Yaskawa INFORM job: OK_R2_O38-47,64(1)(90,180)_HARDO.JBI

/JOB
//NAME OK_R2_O38-47,64(1)(90,180)_HARDO
///FOLDERNAME X4
//POS
///NPOS 800,800,800,27,0,0
///TOOL 0
///POSTYPE PULSE
///PULSE
C00000=-90909,-97924,-91406,-33882,56334,85304
C00001=-91259,-96225,-90754,-33542,56592,85046
C00002=-89195,-70570,-78323,-22025,66185,85062
C00003=-92493,-17269,-45698,-9840,97075,81335
C00004=-91017,-18219,-43079,-10012,95177,81978
C00005=-91017,-18348,-42567,-10003,94801,82008
C00006=-91017,-18513,-41854,-9992,94286,82047
C00007=-91016,-18479,-42013,-9993,94400,82038
C00008=-90999,-21146,-43962,-9991,94233,82058
C00009=-91016,-18479,-42013,-9993,94400,82038
C00010=-92024,-18257,-41848,-9852,94294,81714
C00011=-93307,-17743,-41470,-9670,94175,81298
C00012=-92024,-17970,-43013,-9870,95146,81646
C00013=-103789,-67957,-64906,12961,58029,80477
C00014=-103344,-68399,-64680,12784,57602,80605
C00015=-103344,-68177,-63508,12869,57010,80534
C00016=-103344,-68220,-63718,12855,57117,80546
C00017=-103133,-65270,-62235,12663,57675,80699
C00018=-103344,-68220,-63718,12855,57117,80546
C00019=-102110,-68679,-63945,12230,56831,81014
C00020=-100734,-69291,-64248,11527,56502,81539
C00021=-102110,-68955,-65416,12130,57578,81100
C00022=-83930,-36393,-48077,-21091,64166,86746
C00023=-83530,-35162,-44070,-21603,62556,87219
C00024=-83530,-35090,-42657,-21762,61780,87376
C00025=-83530,-35104,-42903,-21736,61913,87350
C00026=-83323,-32550,-41219,-21780,62224,87371
C00027=-83530,-35104,-42903,-21736,61913,87350
C00028=-84416,-35012,-42843,-21317,61693,87037
C00029=-85758,-34937,-42794,-20674,61360,86560
C00030=-84416,-35012,-42843,-21317,61693,87037
C00031=-98607,9794,-21494,8158,96572,85590
C00032=-98154,8993,-20894,8080,95751,85685
C00033=-98154,8801,-20162,8070,95209,85650
C00034=-98154,8841,-20318,8071,95323,85660
C00035=-98340,6335,-22513,8097,95402,85603
C00036=-98154,8841,-20318,8071,95323,85660
C00037=-97649,8538,-20585,8003,95283,85823
C00038=-96706,8027,-21034,7872,95207,86128
C00039=-97649,8860,-21759,8020,96163,85880
C00040=-91418,16997,-18664,7186,97864,88018
C00041=-81575,50041,17092,-6735,115955,80813
C00042=-84341,50404,17488,-7249,115666,79799
C00043=-84633,49569,18016,-7267,114894,79739
C00044=-84633,49489,18537,-7242,114535,79763
C00045=-84633,49518,18343,-7250,114668,79755
C00046=-84609,54795,24149,-7190,113816,79818
C00047=-84609,54766,24403,-7179,113647,79829
C00048=-84663,51666,20976,-7222,114154,79777
C00049=-84658,51948,21286,-7218,114109,79782
C00050=-84658,51915,21548,-7206,113932,79794
C00051=-84658,51950,21266,-7218,114122,79782
C00052=-84668,56412,26217,-7173,113374,79826
C00053=-84668,56378,26569,-7158,113142,79841
C00054=-84634,53730,23622,-7179,113595,79825
C00055=-84637,55494,23519,-7242,114557,79761
C00056=-81397,31619,-5447,10992,111497,83226
C00057=-81473,32242,-2198,10850,109860,83040
C00058=-81473,31956,-1216,10793,109121,82971
C00059=-81473,32044,-1532,10810,109358,82993
C00060=-81453,37801,4324,10764,108721,82941
C00061=-81453,37706,4697,10744,108448,82916
C00062=-81443,35181,2108,10765,108737,82946
C00063=-81447,36511,1500,10844,109776,83041
C00064=-95159,59700,8174,10738,119151,79045
C00065=-82349,25617,-23576,-8938,79907,82210
C00066=-85481,26023,-25062,-8026,81022,81034
C00067=-85695,25195,-23613,-7939,79706,81051
C00068=-85695,24472,-22838,-7959,78866,81106
C00069=-85695,24604,-22984,-7954,79022,81095
C00070=-85639,26782,-20858,-7986,78839,81125
C00071=-85695,24604,-22984,-7954,79022,81095
C00072=-86173,38935,-12977,-7015,88429,87162
C00073=-85344,38540,-13390,-7315,88547,87404
C00074=-86172,38929,-12971,-7015,88439,87166
C00075=-84007,53583,-39,-17366,95072,84572
C00076=-84007,52813,643,-17337,94292,84683
C00077=-84007,52406,1031,-17322,93863,84745
C00078=-84007,52527,916,-17328,93991,84727
C00079=-84079,50201,-1661,-17319,94351,84652
C00080=-84007,52527,916,-17328,93991,84727
C00081=-84889,52670,1073,-17081,93801,84474
C00082=-85681,52912,1343,-16856,93611,84250
C00083=-84889,53509,304,-17110,94667,84353
C00084=-82262,58897,13828,-12408,108012,82136
C00085=-83953,58737,25467,-6224,116924,79977
C00086=-84346,-10282,-49110,5038,88729,85099
C00087=-83106,-20728,-52489,-22212,92643,80661
C00088=-106659,-18282,-50653,-15937,87636,73637
C00089=-135463,84611,26036,-8427,98138,63561
C00090=-134711,78652,30015,-19475,126025,58919
C00091=-134415,83458,36943,-18891,124399,59387
C00092=-134415,83178,37391,-18788,124001,59464
C00093=-134415,82845,37969,-18663,123504,59559
C00094=-134415,83107,37513,-18763,123898,59484
C00095=-133823,86478,41707,-18417,123218,59859
C00096=-133823,86166,42311,-18294,122713,59953
C00097=-134051,84793,40603,-18428,122994,59806
C00098=-133823,86534,41603,-18437,123307,59843
C00099=-130836,86678,38865,-21284,122414,55409
C00100=-135463,84611,26036,-8427,98138,63561
C00101=-106659,-18282,-50653,-15937,87636,73637
C00102=-89310,-122172,-106686,-13361,50676,45199
C00103=-123165,-113898,-119110,19125,43336,-19368
C00104=-123668,-102412,-109547,19577,43467,-19587
C00105=-131184,63359,57441,15233,67840,-18691
C00106=-122068,78147,74274,12505,69533,-15106
C00107=-122051,87849,89370,12875,65325,-15559
C00108=-122051,89227,92048,12969,64408,-15664
C00109=-122316,85057,86118,12868,65923,-15592
C00110=-122667,82911,83414,12880,66527,-15655
C00111=-122667,83831,85320,12946,65844,-15732
C00112=-122426,86931,89254,12983,65000,-15737
C00113=-122963,79390,78884,12845,67528,-15654
C00114=-130632,64185,60223,15235,66493,-18662
C00115=-131662,58983,54996,15425,67212,-18954
C00116=-131668,55339,42428,14901,72880,-18222
C00117=-146861,-92393,-105699,36485,53490,-27620
C00118=-148000,-101656,-114811,36865,54640,-27702
C00119=-148000,-101656,-114811,36865,54640,-27702
C00120=-148000,-101656,-114811,36865,54640,-27702
C00121=-159496,-161049,-136264,30615,73499,-21221
C00122=-103228,-122632,-133352,-7038,92284,-523
C00123=-103228,-122632,-133352,-7038,92284,-523
C00124=-103228,-124480,-131601,-7026,90271,-411
C00125=-103391,-121920,-131082,-6996,91247,-517
C00126=-103853,-115329,-128981,-6922,93290,-780
C00127=-103391,-120798,-132087,-7006,92433,-583
C00128=-104641,-114737,-130152,-6774,94243,-1084
C00129=-104641,-114737,-130152,-6774,94243,-1084
C00130=-104641,-116137,-129119,-6762,92896,-1012
C00131=-104641,-115940,-129279,-6764,93095,-1023
C00132=-105111,-108950,-126961,-6694,95208,-1287
C00133=-104576,-115792,-130426,-6785,93876,-1044
C00134=-103741,-127928,-135528,-6927,90867,-609
C00135=-103741,-127928,-135528,-6927,90867,-609
C00136=-103741,-127928,-135528,-6927,90867,-609
C00137=-103865,-116944,-129962,-6921,93061,-771
C00138=-103865,-118485,-128547,-6909,91408,-679
C00139=-103865,-118011,-129031,-6913,91946,-709
C00140=-104350,-111197,-126797,-6823,94018,-978
C00141=-103645,-119716,-131347,-6963,92509,-670
C00142=-126331,-111187,-127566,-2170,93341,-7936
C00143=-126314,-110675,-127191,-2173,93374,-7931
C00144=-126314,-111741,-126360,-2171,92316,-7913
C00145=-126314,-111248,-126762,-2172,92816,-7922
C00146=-126152,-104604,-124481,-2216,94828,-7909
C00147=-126314,-111061,-126906,-2173,93001,-7925
C00148=-125902,-111149,-126935,-2263,92984,-7794
C00149=-132196,-109284,-126305,2386,93568,-14490
C00150=-132014,-110397,-125220,2342,92324,-14457
C00151=-132014,-111538,-124094,2340,91046,-14481
C00152=-132014,-110972,-124684,2340,91699,-14468
C00153=-131346,-109003,-124013,2196,92280,-14246
C00154=-132122,-112463,-125993,2364,91740,-14502
C00155=-130696,-128652,-136015,2037,89553,-14081
C00156=-130696,-128652,-136015,2037,89553,-14081
C00157=-134573,-129962,-127961,2886,84044,-15460
C00158=-135247,-123905,-124729,3029,85191,-15657
C00159=-135247,-124242,-122895,3032,83891,-15687
C00160=-135059,-121526,-122583,2986,85086,-15595
C00161=-134621,-115318,-120572,2888,87018,-15405
C00162=-135273,-124345,-124575,3033,84868,-15671
C00163=-101634,-140552,-130463,-4330,80438,-4385
C00164=-100831,-135445,-127742,-4507,81431,-4148
C00165=-100831,-135220,-126147,-4516,80567,-4118
C00166=-100831,-135304,-126661,-4513,80840,-4129
C00167=-101541,-127818,-124438,-4340,83274,-4455
C00168=-100689,-136992,-128168,-4541,80909,-4084
C00169=-101700,-117063,-135109,-4321,95328,-4920
C00170=-101700,-117063,-135109,-4321,95328,-4920
C00171=-107464,-106510,-121453,-3057,92107,-6652
C00172=-105693,-105772,-119256,-3437,91202,-6062
C00173=-105693,-106748,-117862,-3435,89847,-6024
C00174=-105693,-106325,-118509,-3436,90460,-6041
C00175=-104724,-99451,-116018,-3652,92493,-5788
C00176=-105563,-106984,-120499,-3466,91350,-6023
C00177=-97637,-124436,-133710,-5150,90918,-3458
C00178=-101700,-117063,-135109,-4321,95328,-4920
C00179=-101700,-117063,-135109,-4321,95328,-4920
C00180=-113885,-115939,-123860,-1658,88568,-8649
C00181=-113885,-115976,-123799,-1658,88510,-8649
C00182=-113885,-116503,-122835,-1658,87648,-8639
C00183=-113928,-115223,-122529,-1647,88114,-8658
C00184=-114061,-111130,-121156,-1620,89368,-8717
C00185=-113613,-117192,-124203,-1715,88138,-8556
C00186=-77135,-109099,-124316,-9289,94737,2930
C00187=-77964,-100968,-118468,-9143,95217,2626
C00188=-77964,-101677,-117713,-9127,94398,2685
C00189=-77964,-101560,-117850,-9129,94540,2675
C00190=-78928,-97543,-116360,-8967,95572,2290
C00191=-77908,-100245,-119438,-9173,96179,2574
C00192=-71973,-123086,-130703,-10190,92110,4818
C00193=-61369,-106979,-129386,18745,110548,-43775
C00194=-54050,-118433,-122678,29834,105379,-66043
C00195=-54050,-118432,-122677,29849,105379,-66042
C00196=-52380,-128849,-120518,29019,98947,-67079
C00197=-52380,-128559,-118965,28945,98241,-67262
C00198=-52380,-128751,-119946,28990,98681,-67146
C00199=-50245,-132811,-121152,28917,96763,-66805
C00200=-52380,-128751,-119946,28990,98681,-67146
C00201=-49374,-119498,-117890,29381,100712,-65454
C00202=-49135,-119946,-117683,29342,100317,-65463
C00203=-49135,-119959,-116418,29258,99629,-65643
C00204=-49135,-119963,-116925,29289,99902,-65571
C00205=-47420,-122909,-117861,29192,98489,-65269
C00206=-49767,-118756,-118042,29437,101266,-65461
C00207=-58824,-127197,-127906,29549,105900,-67783
C00208=-58824,-127197,-127906,29549,105900,-67783
C00209=-55789,-138532,-125635,28743,98511,-68512
C00210=-54845,-137144,-123724,28738,97781,-68329
C00211=-54845,-136558,-122036,28679,97131,-68490
C00212=-54845,-136878,-122937,28709,97474,-68406
C00213=-52687,-141381,-124200,28678,95380,-68093
C00214=-56052,-135036,-125386,28893,100051,-68223
C00215=-56052,-135036,-125386,28893,100051,-68223
C00216=-54923,-136926,-123517,28734,97796,-68355
C00217=-54923,-136449,-122129,28684,97260,-68488
C00218=-54923,-136715,-122887,28711,97551,-68416
C00219=-52628,-141500,-124230,28677,95326,-68085
C00220=-54923,-138669,-131970,29176,101590,-67387
C00221=-49576,-128334,-132403,27234,106270,-69223
C00222=-44922,-139442,-128392,26353,97465,-69516
C00223=-43106,-142181,-127565,26251,95168,-69348
C00224=-43106,-141292,-125343,26201,94348,-69532
C00225=-43106,-141708,-126356,26223,94717,-69449
C00226=-42222,-150085,-128620,26118,91814,-69764
C00227=-43106,-141708,-126356,26223,94717,-69449
C00228=-58006,-149727,-131155,24086,101568,-78058
C00229=-67130,-160484,-130477,19696,102779,-86761
C00230=-65656,-163702,-131169,20680,100336,-85246
C00231=-25743,-109032,-115433,27145,106620,-70118
C00232=-31386,-185321,-134069,30256,67850,-60806
C00233=-40913,-181249,-136978,30366,76641,-63974
C00234=-31337,-124593,-132531,25311,107075,-53461
C00235=-107165,-96970,-126665,-3187,100215,-6761
C00236=-107165,-106401,-121090,-3121,91950,-6553
C00237=-99006,-123912,-120398,-10471,76789,317
C00238=-104449,-120133,-119195,-8811,77334,-1598
C00239=-136314,-76901,-102772,1273,87959,-12257
C00240=-129245,-75238,-102051,-6216,89043,-4909
C00241=-138081,-104464,-122106,1833,85725,-12838
C00242=-119260,-105046,-123410,-8534,87528,-2432
C00243=-124620,-151805,-134891,-7305,72242,-3267
C00244=-124614,-151414,-134787,-7302,72378,-3273
C00245=-124612,-151215,-134734,-7300,72449,-3276
C00246=-124620,-151805,-134891,-7305,72242,-3267
C00247=-127969,-108981,-129625,-6073,90620,-5362
C00248=-128058,-112032,-130642,-6044,89675,-5344
C00249=-99990,-117497,-120264,-13536,83880,4252
C00250=-95946,-115412,-117807,-14495,84133,5598
C00251=-139069,-101671,-113062,-2900,83618,-8638
C00252=-134512,-124069,-125019,-4259,79673,-7022
C00253=-124704,-125859,-130096,-7035,82535,-3892
C00254=-99313,-127153,-133045,12119,95446,-32872
C00255=-57886,-133831,-130402,29291,103936,-67934
C00256=-55789,-138532,-125635,28743,98511,-68512
C00257=-48693,-117877,-116324,29063,104784,-69163
C00258=-50073,-120833,-117390,28223,106210,-71565
C00259=-68626,-163926,-129258,19114,104295,-87122
C00260=-70376,-133538,-127464,20847,118406,-85282
C00261=-70376,-133538,-127464,20847,118406,-85282
C00262=-57461,-97931,-109353,30188,105270,-63675
C00263=-56121,-79134,-101591,31100,116741,-68778
C00264=-90239,-137211,-122130,21625,111934,-84005
C00265=-78206,-119593,-116830,16675,122083,-90308
C00266=-77714,-101700,-117389,19308,131076,-88387
C00267=-81561,-124200,-134149,21063,125175,-90603
C00268=-103376,-109759,-132308,-3968,97270,-5504
C00269=-101634,-140552,-130463,-4330,80438,-4385
C00270=-110031,-125673,-123303,3182,83425,-15942
C00271=-90641,-116743,-120449,-11075,89773,6751
C00272=-125358,-116095,-120243,-4332,86705,-4548
C00273=-114606,-95150,-113030,-13927,98680,11559
C00274=-109678,-119625,-133746,-14623,99658,13079
C00275=-112326,-124641,-135293,-14185,97639,12436
C00276=-113675,-111285,-124420,-14007,97585,11993
C00277=-113699,-111426,-124467,-14002,97539,11990
C00278=-124004,-129907,-130136,-8507,87303,2218
C00279=-139409,-131326,-130615,456,84743,-11777
C00280=-149006,-99791,-120232,2566,94725,-14751
C00281=-149042,-99754,-120218,2574,94737,-14762
C00282=-144445,-99331,-120062,1565,94748,-13320
C00283=-148134,-92536,-117492,2386,96740,-14437
C00284=-154718,-145008,-134516,3815,80522,-16974
C00285=-155631,-143491,-134098,4008,81086,-17267
C00286=-124045,-119827,-121338,-6126,86009,-1689
C00287=-127884,-116949,-120404,-5328,86643,-2988
C00288=-148100,-95243,-112662,-980,92257,-9671
C00289=-137287,-91556,-109748,-13625,92659,296
C00290=-127829,-127486,-128792,-15513,87749,4031
C00291=-127829,-122446,-134816,-15592,93826,3264
C00292=-125285,-108995,-105645,24533,66859,-22374
C00293=-121876,-100663,-100590,22961,66967,-21017
C00294=-120611,-97454,-98556,22372,66992,-20522
C00295=-120728,-95778,-96365,22498,66572,-20652
C00296=-120611,-97454,-98556,22372,66992,-20522
C00297=-120972,-98646,-98782,22597,66650,-20731
C00298=-119814,-94892,-97816,21908,67582,-20099
C00299=-120972,-98646,-98782,22597,66650,-20731
C00300=-122255,-101873,-100811,23195,66623,-21236
C00301=-125713,-110249,-105850,24792,66512,-22621
C00302=-125414,-109454,-110952,25434,70557,-21724
C00303=-121886,-100912,-105844,23885,70668,-20357
C00304=-120575,-97642,-103795,23303,70688,-19860
C00305=-120636,-96154,-101667,23400,70203,-19982
C00306=-120575,-97642,-103795,23303,70688,-19860
C00307=-121028,-97980,-103315,23548,70382,-20093
C00308=-119871,-93906,-102218,22897,71374,-19458
C00309=-121028,-97980,-103315,23548,70382,-20093
C00310=-122351,-101230,-105354,24132,70373,-20595
C00311=-125908,-109706,-110431,25687,70298,-21973
C00312=-125468,-108852,-114009,26132,73198,-21211
C00313=-121864,-100250,-108878,24604,73277,-19846
C00314=-120523,-96969,-106822,24029,73283,-19350
C00315=-120543,-95651,-104748,24106,72739,-19471
C00316=-120523,-96969,-106822,24029,73283,-19350
C00317=-121096,-97384,-106424,24308,73024,-19616
C00318=-119937,-93066,-105230,23683,74062,-18974
C00319=-121096,-97384,-106424,24308,73024,-19616
C00320=-122450,-100644,-108468,24886,73032,-20117
C00321=-126090,-109173,-113564,26418,72994,-21493
C00322=-126107,-105383,-120588,25792,78658,-20214
C00323=-115870,-101424,-121533,-41206,90180,-3452
C00324=-115851,-106682,-115012,-41260,85065,-1433
C00325=-119242,-98694,-109765,-40357,84214,-2540
C00326=-120508,-95652,-107669,-40003,83867,-2939
C00327=-120512,-93942,-105232,-40036,83383,-2757
C00328=-120508,-95652,-107669,-40003,83867,-2939
C00329=-119976,-95300,-106376,-40178,83625,-2624
C00330=-123146,-93912,-105979,-39274,82602,-3565
C00331=-119976,-95300,-106376,-40178,83625,-2624
C00332=-118706,-98291,-108457,-40527,83992,-2228
C00333=-115305,-106116,-113657,-41413,84900,-1133
C00334=-117529,-113204,-110114,-15038,59483,16836
C00335=-119860,-102582,-104476,-13511,61010,15725
C00336=-120710,-98611,-102232,-12973,61516,15338
C00337=-120712,-96036,-99318,-13028,61058,15391
C00338=-120710,-98611,-102232,-12973,61516,15338
C00339=-120133,-97446,-101425,-13271,61707,15536
C00340=-121539,-92419,-99938,-12330,63118,14842
C00341=-120133,-97446,-101425,-13271,61707,15536
C00342=-119274,-101350,-103659,-13810,61233,15923
C00343=-116924,-111770,-109266,-15331,59803,17031
C00344=-118012,-90030,-113480,-10859,76824,11039
C00345=-121151,-43618,-104634,1145,105190,-4571
C00346=-120753,-40362,-99446,1000,103667,-4481
C00347=-120604,-39041,-97355,946,103057,-4446
C00348=-120606,-40163,-95662,941,101440,-4458
C00349=-120604,-39041,-97355,946,103057,-4446
C00350=-120772,-35445,-95769,1008,103931,-4483
C00351=-120462,-29091,-92658,908,105279,-4391
C00352=-120772,-35445,-95769,1008,103931,-4483
C00353=-120921,-36668,-97839,1062,104577,-4517
C00354=-121319,-39651,-102962,1210,106200,-4605
C00355=-108629,-121399,-122702,-16889,67135,14241
C00356=-115336,-113367,-105488,-19088,53546,18271
C00357=-117865,-102996,-100223,-17109,54980,16930
C00358=-118786,-99066,-98108,-16412,55481,16461
C00359=-118815,-96798,-95161,-16518,54853,16552
C00360=-118786,-99066,-98108,-16412,55481,16461
C00361=-119112,-97264,-98148,-16039,56331,16193
C00362=-118757,-93015,-97035,-15990,57843,16106
C00363=-119112,-97264,-98148,-16039,56331,16193
C00364=-123316,-98367,-98161,-13561,55035,14648
C00365=-126858,-97217,-97820,-11275,54872,13210
C00366=-123316,-98367,-98161,-13561,55035,14648
C00367=-122519,-102389,-100318,-14180,54451,15058
C00368=-120328,-113051,-105701,-15959,52759,16243
C00369=-124093,-110707,-95637,16539,52225,-18162
C00370=-121727,-101468,-90458,14864,53273,-16967
C00371=-120864,-97923,-88367,14268,53637,-16545
C00372=-120864,-95769,-85768,14357,53158,-16613
C00373=-120864,-97923,-88367,14268,53637,-16545
C00374=-120753,-94948,-87925,13988,54838,-16331
C00375=-119636,-91806,-87160,13170,55764,-15745
C00376=-120753,-94948,-87925,13988,54838,-16331
C00377=-121593,-98445,-90034,14553,54501,-16732
C00378=-123889,-107558,-95262,16133,53518,-17861
C00379=-123907,-109460,-104253,15319,57915,-17198
C00380=-120718,-89127,-94408,-93,103364,81793
C00381=-120702,-88967,-86044,-90,98299,81802
C00382=-120714,-92346,-83648,-90,95088,81800
C00383=-120719,-93530,-82604,-90,93837,81800
C00384=-120721,-91291,-79709,-90,93204,81799
C00385=-120719,-93530,-82604,-90,93837,81800
C00386=-120503,-94372,-82680,-81,93451,81873
C00387=-120503,-97134,-83277,-81,92401,81874
C00388=-120503,-94372,-82680,-81,93451,81873
C00389=-120501,-93212,-83739,-81,94699,81873
C00390=-120496,-89894,-86173,-82,97902,81873
C00391=-120512,-90208,-94601,-84,102927,81864
C00392=-120739,-87258,-85833,-92,99047,81789
C00393=-120752,-90752,-83510,-91,95822,81787
C00394=-120758,-91982,-82493,-91,94564,81786
C00395=-120759,-89478,-79257,-91,93861,81786
C00396=-120758,-91982,-82493,-91,94564,81786
C00397=-120462,-95334,-83503,-80,93464,81887
C00398=-120461,-97919,-84058,-79,92477,81888
C00399=-120462,-95334,-83503,-80,93464,81887
C00400=-120460,-94163,-84562,-80,94717,81887
C00401=-120456,-90813,-86994,-80,97935,81887
C00402=-121033,-93279,-128320,140,99068,-4698
C00403=-120997,-110061,-117241,128,83627,-4703
C00404=-120579,-101211,-110995,15,84330,-4566
C00405=-120424,-97983,-108548,-25,84483,-4515
C00406=-120430,-96385,-106046,-24,83763,-4517
C00407=-120424,-97983,-108548,-25,84483,-4515
C00408=-120936,-92390,-106244,111,85940,-4681
C00409=-120538,-86818,-104536,4,87751,-4552
C00410=-120936,-92390,-106244,111,85940,-4681
C00411=-121096,-95373,-108656,154,85891,-4732
C00412=-121527,-103462,-114785,270,85508,-4872
C00413=-75677,-91018,-121004,-38809,104477,-3256
C00414=-86494,-89564,-122641,-29897,102391,-4704
C00415=-121241,-108971,-117698,1136,79653,-4828
C00416=-120728,-99263,-111358,963,80734,-4651
C00417=-120539,-95742,-108880,900,81016,-4587
C00418=-120543,-94296,-106552,902,80326,-4593
C00419=-120539,-95742,-108880,900,81016,-4587
C00420=-120728,-93992,-107595,961,81127,-4647
C00421=-120728,-90301,-106424,959,82303,-4638
C00422=-120728,-93992,-107595,961,81127,-4647
C00423=-121024,-97533,-112143,1058,82109,-4735
C00424=-121551,-107098,-118478,1235,81100,-4915
C00425=-121569,-100080,-124444,1231,88376,-4850
C00426=-117898,-83225,-110918,-12916,113641,67504
C00427=-119870,-90654,-110250,-12481,109228,67312
C00428=-120686,-93336,-109842,-12338,107519,67211
C00429=-120688,-92183,-107571,-12276,106730,67294
C00430=-120686,-93336,-109842,-12338,107519,67211
C00431=-120163,-91649,-109473,-12395,108219,67318
C00432=-121681,-97188,-111137,-12239,106219,67001
C00433=-120163,-91649,-109473,-12395,108219,67318
C00434=-119359,-88923,-109851,-12543,109932,67413
C00435=-117416,-81399,-110449,-12994,114344,67589
C00436=-120617,-94125,-108136,8857,121741,88541
C00437=-120616,-94449,-107526,8800,121205,88496
C00438=-136098,-107181,-107429,16269,112846,84409
C00439=-120444,-95183,-107742,8816,120947,88541
C00440=-119761,-91680,-105499,9024,121288,-74873
C00441=-120616,-95784,-105179,-19399,105655,65758
C00442=-120617,-94769,-108163,-19676,107886,65380
C00443=-121686,-93853,-106574,-24019,104588,57765
C00444=-120617,-92780,-110041,-24421,107344,57569
C00445=-120617,-90665,-112384,-24828,109654,57058
C00446=-120619,-82046,-117525,-26421,116533,55408
C00447=-120645,-81988,-112872,-3577,88664,15070
C00448=-120614,-96077,-90479,12976,48732,-14983
C00449=-120612,-93911,-81283,13967,44304,-15634
C00450=-120612,-93390,-79613,14157,43566,-15753
C00451=-121252,-93346,-79166,14714,43437,-16096
C00452=-121500,-95247,-79374,15137,42660,-16355
C00453=-120782,-94947,-80724,14317,43483,-15851
C00454=-120611,-93982,-79716,14233,43318,-15795
C00455=-120612,-95725,-83890,13821,44941,-15536
C00456=-121326,-94847,-83951,14224,45559,-15784
C00457=-120613,-94980,-84633,13612,45776,-15407
C00458=-120613,-95388,-86250,13438,46540,-15293
C00459=-120616,-96933,-104006,-5046,49827,-739
C00460=-120616,-97132,-103061,-5097,49146,-704
C00461=-120617,-95323,-101728,-5088,49256,-711
C00462=-120871,-100699,-104338,-4972,48087,-759
C00463=-120795,-98262,-101888,-5054,47837,-712
C00464=-120618,-95198,-103493,-5003,50401,-770
C00465=-121122,-95129,-103646,-4600,50501,-986
C00466=-120617,-97030,-104927,-5009,50342,-766
C00467=-120617,-96757,-105844,-4959,51045,-801
C00468=-120618,-92718,-112658,-4589,57292,-1090
C00469=-108098,-105677,-132023,-7461,89264,328
C00470=-80455,-75739,-120669,-16714,100968,7375
C00471=-97258,-84752,-105297,-10869,90674,3530
C00472=-97358,-86422,-102930,-10833,88387,3696
C00473=-97424,-86715,-102018,-10818,87679,3736
C00474=-97216,-90521,-102980,-10875,86365,3919
C00475=-97404,-84940,-102216,-10822,88698,3655
C00476=-120617,-94266,-106774,-4665,84598,-3614
C00477=-111454,-84543,-103018,-13521,90962,7073
C00478=-109783,-86139,-104921,-12729,90791,5985
C00479=-106092,-100123,-116923,-13597,91547,7106
C00480=-102052,-116072,-128299,-14497,91044,8487
C00481=-91007,-121504,-125767,-15485,91359,21712
C00482=-120613,-95050,-86060,-3557,95049,80550
C00483=-120612,-93945,-81838,-3544,93023,80607
C00484=-121155,-91942,-79314,-3616,92478,80448
C00485=-120652,-94806,-81837,-3543,92579,80606
C00486=-120610,-90975,-79567,-3544,93151,80605
C00487=-150255,-82598,-75582,-4413,93505,70504
C00488=-122384,-91795,-77981,-11848,92227,69969
C00489=-120612,-93489,-79991,-12120,92904,70125
C00490=-120613,-94640,-84016,-12161,94749,69944
C00491=-120614,-96377,-93023,-12320,99298,69491
C00492=-120644,-125570,-121052,6784,67869,5403
C00493=-120615,-96622,-98748,12572,58745,-14095
C00494=-120615,-96643,-96984,12717,57674,-14222
C00495=-127606,-89142,-93330,20657,62312,-19456
C00496=-120926,-99715,-97034,13118,56212,-14526
C00497=-120613,-97817,-97899,12721,57634,-14225
C00498=-120615,-96818,-95655,-6616,54391,-866
C00499=-120615,-97044,-96976,-6561,55085,-910
C00500=-112093,-90513,-93108,-22044,58833,17349
C00501=-120615,-96644,-96112,-9528,53512,9485
C00502=-120615,-96653,-97679,-9416,54459,9397
C00503=-120616,-95373,-105489,-8868,59856,8934
C00504=-117333,-91440,-108817,-14098,83709,30265
C00505=-112347,-94381,-87846,-22750,99580,64599
C00506=-112329,-92021,-78548,-22454,95406,65402
C00507=-115628,-91274,-75119,-22621,92902,64661
C00508=-117255,-90241,-73175,-22718,91835,64269
C00509=-117028,-88603,-73220,-22719,92705,64185
C00510=-116923,-92272,-75451,-22697,92259,64308
C00511=-120553,-90828,-77383,15099,94128,70510
C00512=-120613,-90885,-77384,15804,94030,70628
C00513=-123770,-105111,-82751,16580,84167,79857
C00514=-124886,-104010,-85216,16560,86394,79763
C00515=-120613,-94284,-84162,15892,96365,70931
C00516=-120614,-95920,-93129,16139,100869,71526
C00517=-120649,-92160,-111225,3199,84919,49711
C00518=-120616,-97604,-99172,-11891,40402,23254
C00519=-120614,-96911,-90603,-13253,35598,24030
C00520=-120614,-96763,-89737,-13401,35153,24111
C00521=-121291,-96342,-89250,-12683,34963,23744
C00522=-119113,-97762,-90324,-15090,35268,24978
C00523=-120705,-99580,-90146,-13704,33974,24279
C00524=-121588,-95238,-86691,-12692,33949,23762
C00525=-127502,-77730,-88040,1756,56127,19882
C00526=-125086,-93679,-98074,150,54079,20822
C00527=-120613,-95818,-85653,-14108,33181,24494
C00528=-120615,-97479,-97669,-6545,55280,-923
C00529=-121580,-96410,-96097,-5967,54791,-1285
C00530=-120928,-100587,-97757,-6468,53722,-953
C00531=-120613,-98670,-98620,-6548,55254,-920
C00532=-120615,-96854,-96360,-6584,54805,-893
C00533=-120615,-97074,-97513,-6537,55399,-931
C00534=-114077,-92170,-94328,-19163,57465,15491
C00535=-120615,-97626,-97578,-9481,53904,9448
C00536=-120636,-112691,-117418,-8831,59265,10492
C00537=-120617,-94408,-109491,-7961,65698,13071
C00538=-120616,-97035,-102174,-8375,59902,13490
C00539=-120616,-97254,-100452,-8474,58742,13580
C00540=-120616,-96110,-99125,-8495,58514,13598
C00541=-120614,-98453,-101360,-8481,58685,13585
C00542=-119727,-100186,-100479,-9138,57364,14041
C00543=-120617,-96158,-99373,-8483,58642,13587
C00544=-120616,-97215,-100721,-8458,58926,13566
C00545=-120616,-96978,-102436,-8360,60091,13476
C00546=-120617,-94247,-109716,-7948,65917,13056
C00547=-120616,-96445,-103082,5252,59171,-13430
C00548=-120615,-96888,-94956,5569,53965,-13694
C00549=-120614,-96711,-93127,5642,52935,-13750
C00550=-120614,-96618,-92386,5672,52529,-13773
C00551=-119756,-94067,-91753,5051,53390,-13370
C00552=-120525,-97964,-94062,5589,52861,-13717
C00553=-120614,-96681,-92800,5656,52750,-13760
C00554=-120614,-96709,-92988,5648,52851,-13755
C00555=-120614,-96767,-93400,5632,53074,-13742
C00556=-120614,-96843,-94134,5603,53484,-13720
C00557=-120615,-96977,-95945,5531,54526,-13664
C00558=-120616,-97003,-101109,6851,58481,-13557
C00559=-120615,-97139,-99377,6934,57353,-13629
C00560=-120615,-97164,-98672,6968,56909,-13657
C00561=-119756,-94335,-97933,6375,57832,-13263
C00562=-120570,-98373,-100300,6912,57283,-13615
C00563=-120615,-97165,-99156,6946,57204,-13638
C00564=-120616,-97129,-99856,6912,57651,-13610
C00565=-120616,-96964,-101578,6829,58787,-13537
C00566=-120617,-96349,-105255,7716,61917,-13386
C00567=-120616,-96771,-103611,7804,60699,-13471
C00568=-120616,-96905,-102940,7840,60222,-13505
C00569=-119756,-93851,-102113,7266,61195,-13116
C00570=-120602,-97980,-104523,7800,60639,-13470
C00571=-120616,-96844,-103353,7819,60505,-13485
C00572=-120616,-96699,-104019,7783,60985,-13451
C00573=-120617,-96245,-105652,7696,62212,-13366
C00574=-120618,-92150,-112439,7334,68442,-12961
C00575=-130920,-122289,-127601,-23263,76296,33617
C00576=-126647,-121486,-124764,-14921,71090,19914
C00577=-118673,-117816,-113052,-9081,54805,1270
C00578=-119719,-97166,-102733,-8035,58912,525
C00579=-118944,-92090,-109805,-27006,83902,36269
C00580=-120616,-93914,-111601,-26462,83549,35758
C00581=-120617,-94475,-108119,-24525,75199,30020
C00582=-120618,-90011,-113520,-23738,94905,43572
C00583=-120617,-93534,-109718,-22404,79768,31867
C00584=-120617,-93028,-110386,-24696,84592,28860
C00585=-120617,-93859,-109223,-24523,82429,27907
C00586=-120617,-95217,-106728,-22357,73913,21133
C00587=-120616,-96198,-104144,-16550,64688,11231
C00588=-120616,-97587,-102867,-7505,58697,196
C00589=-120615,-98378,-102979,677,57412,-8649
C00590=-120615,-98092,-104435,2505,58558,-10610
C00591=-120615,-97859,-104607,2041,58746,-10113
C00592=-120615,-97689,-104685,1580,58853,-9618
C00593=-120615,-97267,-104663,-2078,59079,-5700
C00594=-122185,-96113,-104438,-1107,59504,-6297
C00595=-124417,-94235,-103728,259,60020,-7133
C00596=-120617,-96195,-105273,-2057,60007,-5718
C00597=-120617,-95777,-106468,-2039,60956,-5736
C00598=-120690,-30346,-78642,22937,64170,-21118
C00599=-120690,-30346,-78642,22937,64170,-21118
C00600=-98469,-5770,-79404,6171,73775,-13621
C00601=-73961,-64832,-115099,-11040,66386,-6438
C00602=-152983,-151482,-105999,63266,53723,19798
C00603=-133395,-32083,-56059,41211,61963,37621
C00604=-138234,23065,45169,67508,45202,44915
C00605=-136781,30072,55747,70235,43147,43411
C00606=-136213,33214,60449,71542,42329,42699
C00607=-136213,31591,57334,70422,42710,43384
C00608=-136788,30891,57778,71075,42855,42892
C00609=-134893,29619,56778,71118,41623,43172
C00610=-133284,25640,52793,70642,40733,43707
C00611=-131869,22445,49655,70246,39929,44150
C00612=-132436,19576,45433,69035,40713,44782
C00613=-133889,13007,35719,66469,42691,46136
C00614=-120930,8852,32410,71146,24358,44597
C00615=-120056,16713,42856,76185,23038,42237
C00616=-120570,20810,47735,78353,23157,41125
C00617=-120179,17981,45384,78314,22894,41190
C00618=-119718,18730,44666,76295,22791,42223
C00619=-125399,29317,56132,80433,26238,39500
C00620=-125034,24898,50699,78244,26224,40637
C00621=-126001,16678,39521,73266,27604,43020
C00622=-110893,28996,24386,6920,61269,70362
C00623=-121937,-147756,-98721,13314,47766,64479
C00624=-71720,-152863,-104081,-12596,70757,83485
C00625=-71720,-152863,-104081,-12596,70757,83485
C00626=-91982,-28216,-51992,2303,92813,79298
C00627=-105745,54824,-16277,12342,106777,76346
C00628=-79811,47197,33770,-5226,114025,80115
C00629=-80023,42119,31306,-5246,112923,80086
C00630=-80397,41231,31844,-5317,112121,79984
C00631=-80109,39795,28796,-5290,113266,80037
C00632=-80112,42618,33014,-5241,112126,80089
C00633=-81014,41143,31800,-5517,112061,79755
C00634=-81200,40698,29696,-5625,113108,79635
C00635=-82013,41869,30925,-5879,112897,79339
C00636=-81757,29065,16922,-5439,108904,79311
C00637=-82874,29136,16993,-5696,108820,78911
C00638=-83189,43833,33118,-6256,112463,78920
C00639=-80599,47195,33767,-5484,113974,79819
C00640=-80608,45992,24153,-5781,119246,79546
C00641=-80156,46426,18785,-6968,101557,41119
C00642=-78753,47274,23775,-10662,32517,-78562
C00643=-79428,-41610,-51646,-9616,33163,-79071
C00644=-79413,-40970,-42943,-11157,28217,-78271
C00645=-79779,-35257,-36372,-11029,27079,-78324
C00646=-81991,-26459,-36295,-2567,38667,-80402
C00647=-79917,-33213,-35108,-10725,27328,-78472
C00648=-79914,-35155,-35130,-11097,26361,-78286
C00649=-83153,-26286,-36175,-1364,38653,-81015
C00650=-81501,-33436,-35517,-8333,27283,-79626
C00651=-82704,-33725,-35707,-6541,27141,-80488
C00652=-84536,-24696,-36395,719,41193,-81637
C00653=-85703,-24509,-36263,1843,41226,-82218
C00654=-83984,-33203,-37030,-4447,28135,-81499
C00655=-80764,-40975,-42948,-9214,28047,-79206
C00656=-80778,-41615,-51650,-7929,33019,-79872
C00657=-86790,-31694,-78031,7959,81796,-79340
C00658=-86790,-31694,-78031,7959,81796,54010
C00659=-85481,26023,-25062,-8026,81022,81034
C00660=-85601,25422,-23671,-8007,79839,81046
C00661=-84918,26463,-20904,-8350,78751,81327
C00662=-84396,34572,-13203,-16967,82171,79029
C00663=-84396,34572,-13203,-16967,82171,79029
C00664=-86241,53458,1953,-14539,94111,75660
C00665=-83535,64450,13715,-20994,99928,87619
C00666=-86164,73511,21600,-12190,104413,87957
C00667=-86834,68614,15196,-6594,103697,88880
C00668=-86834,68614,15196,-6594,103697,88880
C00669=-86265,58182,4340,-6215,98305,89490
C00670=-84918,26463,-20904,-8350,78751,81327
C00671=-84270,25392,-25849,-8593,81276,81352
C00672=-83330,-46575,-52890,-13958,55049,-41505
C00673=-86193,-52033,-54165,-20785,79907,1804
C00674=-87571,-35325,-52921,-25788,81678,348
C00675=-87508,-34952,-39783,-27132,74543,196
C00676=-104644,32154,27534,4448,60513,72731
C00677=-93805,201,18674,23355,11914,69008
C00678=-93808,216,18686,23365,11915,69004
C00679=-93810,222,18691,23369,11915,69002
C00680=-93638,2355,20486,22861,11860,69245
C00681=-93955,-2017,16089,22978,12371,69170
C00682=-93808,210,18682,23363,11914,69005
C00683=-93806,198,18671,23357,11914,69008
C00684=-93804,186,18662,23351,11913,69011
C00685=-93802,180,18657,23347,11913,69012
C00686=-93799,166,18644,23338,11912,69017
C00687=-93810,232,18700,23265,11906,69051
C00688=-93813,246,18712,23275,11907,69047
C00689=-94451,684,18996,25087,12134,68175
C00690=-93990,-1863,16961,23823,11950,68785
C00691=-93814,-607,16661,21825,12670,69707
C00692=-100120,3293,21094,39224,14315,61321
C00693=-100936,-4761,10472,35572,16592,62958
C00694=-101724,-18723,-6868,31140,19848,65000
C00695=-104644,32154,27534,4448,60513,72731
C00696=-81813,-56841,-53371,-53266,50302,14082
C00697=-60380,-131230,-84967,-114894,34586,40161
C00698=-75788,-111312,-115723,-41491,75595,63087
C00699=-90161,-54224,-109841,7916,106787,80704
C00700=-89492,4607,-58591,7657,105439,80800
C00701=-89900,18802,-35938,9766,95357,80687
C00702=-83481,65005,13429,-9056,119285,78997
C00703=-83752,59141,12946,-8828,116574,79122
C00704=-105122,63991,30490,2309,126100,76457
C00705=-105343,61862,26796,2259,127285,76391
C00706=-85852,59503,13361,-9003,116292,78389
C00707=-84859,64061,16437,-8959,116837,78702
C00708=-84733,23156,-31643,-6898,102580,79911
C00709=-89806,-37631,-52942,13196,44828,72538
C00710=-94750,-32934,-45091,18174,44929,69862
C00711=-94288,-25470,-35130,18528,42645,69603
C00712=-107305,-33153,-35053,31246,31625,63156
C00713=-107702,-34958,-34985,32523,30946,62498
C00714=-97590,-24051,-34127,21303,43547,68126
C00715=-95242,-30076,-40811,18964,43932,69406
C00716=-95187,-81119,-79791,20309,40550,69551
C00717=-79732,-39015,-61878,-9776,73483,77661
C00718=-79685,-36342,-57499,-9860,72185,77784
C00719=-87087,-35830,-57170,-6595,71518,75302
C00720=-87087,-35830,-57170,-6595,71518,75302
C00721=-90742,-7826,-43743,-2271,93476,74111
C00722=-90914,1844,-37212,-1728,100816,78743
C00723=-95897,12563,-27941,8521,106941,79054
C00724=-92202,11038,-29312,8242,106650,80256
C00725=-92202,11038,-29312,8242,106650,80256
C00726=-93396,-25996,-53787,10938,81976,79329
C00727=-79685,-36342,-57499,-9860,72185,77784
C00728=-79400,-36667,-60385,-9905,73804,77748
C00729=-81287,-73482,-80856,-9429,67353,77616
C00730=-79535,-70349,-76672,-10284,66612,78310
C00731=-88732,-69497,-76162,-6083,65818,75025
C00732=-88732,-69497,-76162,-6083,65818,75025
C00733=-90662,-45473,-68546,-4673,86051,73788
C00734=-98683,-18642,-53546,6653,105150,72806
C00735=-103276,-16438,-50778,15365,106646,73034
C00736=-98885,-19031,-52697,15020,105742,74408
C00737=-98885,-19031,-52697,15020,105742,74408
C00738=-99083,-47180,-68555,16074,86488,72763
C00739=-79535,-70349,-76672,-10284,66612,78310
C00740=-79862,-72759,-79630,-10096,67144,78145
C00741=-79862,-70265,-89965,-9669,74677,77521
C00742=-106636,9561,-40732,-8334,61658,77698
C00743=-105745,52807,-15764,12246,105454,76208
C00744=-120157,82254,53851,-8462,118881,68276
C00745=-120764,76019,49190,-8631,118486,68068
C00746=-120545,72963,46863,-8548,118376,68166
C00747=-121013,73553,46157,-8768,119052,67924
C00748=-120677,76096,50452,-8536,117766,68159
C00749=-121226,74496,48762,-8737,117926,67935
C00750=-121277,74331,46343,-8885,119308,67802
C00751=-123087,79936,53120,-9346,117831,67212
C00752=-122088,74841,49080,-9011,117811,67607
C00753=-123278,77975,52864,-9325,116969,67212
C00754=-123162,86054,59807,-9277,116864,67267
C00755=-123114,53430,10385,-1251,116221,68203
C00756=-136323,52272,9545,44589,64919,61463
C00757=-139783,-33179,-13184,69240,48192,46182
C00758=-137611,-28365,-6875,70201,46216,45730
C00759=-136968,-25802,-3994,70545,45624,45564
C00760=-136770,-25555,-2359,71345,45178,45070
C00761=-137559,-27867,-5282,70853,45921,45309
C00762=-131841,-32977,-8690,70719,41910,45942
C00763=-131975,-36416,-12130,70369,42121,46140
C00764=-134147,-41542,-18435,69427,44030,46529
C00765=-141128,-29133,-31085,43489,44991,50173
C00766=-145944,-19375,-16364,60085,47488,49165
C00767=-145724,-16199,-12904,60405,47092,48951
C00768=-146072,-18893,-14822,60688,47208,48761
C00769=-145286,-17068,-12207,60970,46372,48581
C00770=-149468,-6849,-5739,61336,49653,48312
C00771=-146980,-8744,-14162,48811,51872,51880
C00772=-141391,-26070,-33699,44316,51156,54843
C00773=-135350,-43982,-50251,40364,49000,57185
C00774=-135985,2271,-36804,-9338,77862,64370
C00775=-130949,74091,43956,-19987,113167,60546
C00776=-132080,69549,41488,-20064,112128,60294
C00777=-132880,68865,42086,-20096,111257,60142
C00778=-132541,67844,41901,-19973,110951,60327
C00779=-132116,69898,43068,-19947,111372,60417
C00780=-135736,79269,54433,-20274,108439,59549
C00781=-135060,80104,54141,-20241,109178,59676
C00782=-133923,84725,56898,-20139,110093,59949
C00783=-137379,33195,-5040,-12355,95090,61475
C00784=-141075,-6060,-32928,-6165,69436,63043
C00785=-141075,-2977,-40411,-5973,75592,62734
C00786=-98744,-40754,-67548,-10182,73737,65749
C00787=-77897,36380,-16593,-16424,103812,69919
C00788=-77068,57839,11191,-15964,106904,70080
C00789=-79558,60641,16966,-13373,108460,69494
C00790=-80702,59225,13666,-4367,108593,79878
C00791=-80613,55459,9814,7293,107022,88327
C00792=-74695,56150,10593,6946,106416,90257
C00793=-73933,56289,10752,6898,106334,90508
C00794=-73561,55782,10184,6877,106395,90634
C00795=-74053,58573,11706,6929,106928,90501
C00796=-86051,35712,-26077,8385,119323,87373
C00797=-98744,-40754,-67548,-10182,73737,65749
C00798=-125690,-78122,-87562,-13631,67908,68588
C00799=-2173,-78122,-87562,-13631,67908,68588
BC00000=277590,692280,168144
BC00001=277590,750776,168144
BC00002=277590,762994,168144
BC00003=277590,762994,168144
BC00004=277590,762994,168143
BC00005=277590,762994,168143
BC00006=277590,762994,168143
BC00007=277590,762994,168142
BC00008=277590,762994,168142
BC00009=277590,762994,168142
BC00010=277590,762994,168142
BC00011=277590,762994,168142
BC00012=277590,762994,168142
BC00013=277590,762994,168142
BC00014=277590,762994,168142
BC00015=277590,762994,168142
BC00016=277590,762994,168142
BC00017=277590,762994,168142
BC00018=277590,762994,168142
BC00019=277590,762994,168142
BC00020=277590,762994,168142
BC00021=277590,762994,168142
BC00022=277590,762994,168142
BC00023=277590,762994,168142
BC00024=277590,762994,168142
BC00025=277590,762994,168142
BC00026=277590,762994,168142
BC00027=277590,762994,168142
BC00028=277590,762994,168142
BC00029=277590,762994,168142
BC00030=277590,762994,168142
BC00031=277590,762994,168142
BC00032=277590,762994,168142
BC00033=277590,762994,168142
BC00034=277590,762994,168141
BC00035=277590,762994,168141
BC00036=277590,762994,168141
BC00037=277590,762994,168141
BC00038=277590,762994,168141
BC00039=277590,762994,168141
BC00040=277590,762994,168141
BC00041=274757,787027,149092
BC00042=274757,787027,149092
BC00043=274757,787027,149090
BC00044=274757,787027,149090
BC00045=274757,787027,149090
BC00046=274757,787027,149090
BC00047=274757,787027,149090
BC00048=274757,787027,149090
BC00049=274757,787027,149090
BC00050=274757,787027,149090
BC00051=274757,787027,149090
BC00052=274757,787027,149090
BC00053=274757,787027,149090
BC00054=274757,787027,149090
BC00055=274757,787027,149090
BC00056=274757,787027,149090
BC00057=274757,787027,149090
BC00058=274757,787027,149090
BC00059=274757,787027,149090
BC00060=274757,787027,149090
BC00061=274757,787027,149090
BC00062=274757,787027,149090
BC00063=274757,787027,149090
BC00064=307296,787027,31119
BC00065=278551,787027,4009
BC00066=278551,787027,4009
BC00067=278551,787027,4005
BC00068=278551,787027,4005
BC00069=278551,787027,4005
BC00070=278551,787027,4005
BC00071=278551,787027,4005
BC00072=278551,787026,4004
BC00073=278551,787026,4004
BC00074=278551,787026,4002
BC00075=278551,787026,4002
BC00076=278551,787026,4002
BC00077=278551,787026,4002
BC00078=278551,787026,4002
BC00079=278551,787026,4002
BC00080=278551,787026,4002
BC00081=278551,787026,4002
BC00082=278551,787026,4002
BC00083=278551,787026,4002
BC00084=276870,787567,79557
BC00085=275390,788044,146099
BC00086=277590,791707,168144
BC00087=277590,791707,168144
BC00088=277590,791707,168144
BC00089=337074,760417,53
BC00090=337074,815057,24896
BC00091=337074,815057,53
BC00092=337074,815057,53
BC00093=337074,815057,53
BC00094=337074,815057,53
BC00095=337074,815057,53
BC00096=337074,815057,53
BC00097=337074,815057,53
BC00098=337074,815057,53
BC00099=337074,815057,53
BC00100=337074,780859,53
BC00101=277590,791707,168144
BC00102=277590,719585,168144
BC00103=96859,683802,308578
BC00104=96859,755769,293742
BC00105=128715,819724,308578
BC00106=128715,834124,308578
BC00107=128715,834124,308578
BC00108=128715,834124,308578
BC00109=128715,834124,308578
BC00110=128715,834124,308578
BC00111=128715,834124,308578
BC00112=128715,834124,308578
BC00113=128715,834124,308578
BC00114=128715,819724,308578
BC00115=128715,819724,308578
BC00116=128715,819724,308578
BC00117=128715,755769,293742
BC00118=128715,683802,308578
BC00119=128715,683802,1074810
BC00120=128715,683802,1074810
BC00121=10701,883002,1074810
BC00122=2462,1013180,1073459
BC00123=106,1014076,1058465
BC00124=106,1014076,1058465
BC00125=106,1014076,1058465
BC00126=106,1014076,1058465
BC00127=106,1014076,1058465
BC00128=75740,998026,1061993
BC00129=76500,998506,1056750
BC00130=76500,998506,1056750
BC00131=76500,998506,1056750
BC00132=76500,998506,1056750
BC00133=76500,998506,1056750
BC00134=76500,998506,1056750
BC00135=62326,958870,1056750
BC00136=67570,962518,1021274
BC00137=67570,962518,1021274
BC00138=67570,962518,1021274
BC00139=67570,962518,1021274
BC00140=67570,962518,1021271
BC00141=67570,962518,1021274
BC00142=67570,962518,1021274
BC00143=67570,962518,1021274
BC00144=67570,962518,1021274
BC00145=67570,962518,1021274
BC00146=67570,962518,1021274
BC00147=67570,962518,1021274
BC00148=145480,943896,1073360
BC00149=166821,969292,1072076
BC00150=166821,969292,1072076
BC00151=166821,969292,1072076
BC00152=166821,969292,1072076
BC00153=166821,969292,1072076
BC00154=166821,969292,1072076
BC00155=166820,969293,1072075
BC00156=274128,961901,1072075
BC00157=274128,961901,1072075
BC00158=274128,961901,1072075
BC00159=274128,961901,1072075
BC00160=274128,961901,1072075
BC00161=274128,961901,1072075
BC00162=274128,961901,1072075
BC00163=274128,961901,1072075
BC00164=274128,961901,1072071
BC00165=274128,961901,1072071
BC00166=274128,961901,1072071
BC00167=274128,961901,1072071
BC00168=274128,961901,1072071
BC00169=274128,961901,1072071
BC00170=253787,895567,1072071
BC00171=253787,895567,1066387
BC00172=253787,895567,1066387
BC00173=253787,895567,1066387
BC00174=253787,895567,1066387
BC00175=253787,895567,1066387
BC00176=253787,895567,1066387
BC00177=253787,895567,1066387
BC00178=332690,882659,1072071
BC00179=352776,943841,1062049
BC00180=352776,943841,1056120
BC00181=352776,943841,1056120
BC00182=352776,943841,1056120
BC00183=352776,943841,1056120
BC00184=352776,943841,1056120
BC00185=352776,943841,1056120
BC00186=352776,943841,1056120
BC00187=352776,943841,1056120
BC00188=352776,943841,1056120
BC00189=352776,943841,1056120
BC00190=352776,943841,1056120
BC00191=352776,943841,1056120
BC00192=352776,943841,1056120
BC00193=310169,911968,1073469
BC00194=291623,911782,1074972
BC00195=268902,904998,1073205
BC00196=268902,904998,1073205
BC00197=268902,904998,1073205
BC00198=268902,904998,1073205
BC00199=268902,904998,1073205
BC00200=268902,904998,1073205
BC00201=320878,904998,1073205
BC00202=320878,904998,1073205
BC00203=320878,904998,1073205
BC00204=320878,904998,1073205
BC00205=320878,904998,1073205
BC00206=320878,904998,1073205
BC00207=320878,904998,1073205
BC00208=213337,904998,1073205
BC00209=213337,904998,1068795
BC00210=213337,904998,1068795
BC00211=213337,904998,1068795
BC00212=213337,904998,1068795
BC00213=213337,904998,1068795
BC00214=213337,904998,1068795
BC00215=170757,904998,1068795
BC00216=170757,904998,1068795
BC00217=170757,904998,1068795
BC00218=170757,904998,1068795
BC00219=170757,904998,1068795
BC00220=170757,904998,1068795
BC00221=193221,1067506,1068795
BC00222=193221,1067506,1068795
BC00223=193221,1067506,1068795
BC00224=193221,1067506,1068795
BC00225=193221,1067506,1068795
BC00226=193221,1067506,1068795
BC00227=193221,1067506,1068795
BC00228=199711,1067506,1068794
BC00229=207788,1067506,1068792
BC00230=207788,1067506,1068790
BC00231=207788,1067506,1068792
BC00232=207788,1067506,1068792
BC00233=207788,1067506,1068792
BC00234=207788,1067506,1073587
BC00235=282406,880495,1068555
BC00236=282406,880495,1066387
BC00237=282404,880494,1066387
BC00238=282404,880494,1066387
BC00239=282404,880494,1066387
BC00240=282404,880494,1066387
BC00241=282404,880494,1066387
BC00242=100678,973416,1072339
BC00243=113353,1001451,1072339
BC00244=107557,1002422,1072440
BC00245=36539,1014323,1073683
BC00246=30635,1015327,1073683
BC00247=112239,958761,1072440
BC00248=388770,864829,1072440
BC00249=395574,924315,1072438
BC00250=396601,933289,1072438
BC00251=396601,933289,1072438
BC00252=396601,933289,1072438
BC00253=396601,933289,1072438
BC00254=316599,920939,1070848
BC00255=213337,904998,1068795
BC00256=213337,904998,1068795
BC00257=213337,904998,1068795
BC00258=213337,904998,1068795
BC00259=213337,904998,1068795
BC00260=213337,904998,1068795
BC00261=327385,904998,1068795
BC00262=316881,884304,1068795
BC00263=316881,884304,1068795
BC00264=316881,884304,1068795
BC00265=316881,884304,1068795
BC00266=316881,884304,1068795
BC00267=316098,887435,1068795
BC00268=274128,953808,1072075
BC00269=274128,961901,1072075
BC00270=274129,961901,1072073
BC00271=274129,961901,1072073
BC00272=274129,961901,1072073
BC00273=274129,961901,1072073
BC00274=274129,961901,1072073
BC00275=191184,974268,1072073
BC00276=191184,974268,1072073
BC00277=191184,974268,1072073
BC00278=191184,974268,1072073
BC00279=191184,974268,1072073
BC00280=191184,974268,1072073
BC00281=191184,974268,1072073
BC00282=181213,974268,1072073
BC00283=181213,974268,1072073
BC00284=181213,974268,1072073
BC00285=102087,963066,1072073
BC00286=102087,963066,1072073
BC00287=102087,963066,1072073
BC00288=102087,963066,1072073
BC00289=102087,963066,1072073
BC00290=102087,963066,1072070
BC00291=124233,740604,1070750
BC00292=168854,844547,1075175
BC00293=168854,844547,1075175
BC00294=168854,844547,1075175
BC00295=168854,844547,1075175
BC00296=168854,844547,1075175
BC00297=168854,844547,1075175
BC00298=168854,844547,1075175
BC00299=168854,844547,1075175
BC00300=168854,844547,1075175
BC00301=168854,844547,1075175
BC00302=125556,866811,1075175
BC00303=125556,866811,1075175
BC00304=125556,866811,1075175
BC00305=125556,866811,1075175
BC00306=125556,866811,1075175
BC00307=125556,866811,1075175
BC00308=125556,866811,1075175
BC00309=125556,866811,1075175
BC00310=125556,866811,1075175
BC00311=125556,866811,1075175
BC00312=94030,883389,1075175
BC00313=94030,883389,1075175
BC00314=94030,883389,1075175
BC00315=94030,883389,1075175
BC00316=94030,883389,1075175
BC00317=94030,883389,1075175
BC00318=94030,883389,1075175
BC00319=94030,883389,1075175
BC00320=94030,883389,1075175
BC00321=94030,883389,1075175
BC00322=94030,883389,1075175
BC00323=254016,900546,1075175
BC00324=254016,900546,1075175
BC00325=254016,900546,1075175
BC00326=254016,900546,1075175
BC00327=254016,900546,1075175
BC00328=254016,900546,1075175
BC00329=254016,900546,1075175
BC00330=254016,900546,1075175
BC00331=254016,900546,1075175
BC00332=254016,900546,1075175
BC00333=254016,900546,1075175
BC00334=131751,862217,1075175
BC00335=131751,862217,1075175
BC00336=131751,862217,1075175
BC00337=131751,862217,1075175
BC00338=131751,862217,1075175
BC00339=131751,862217,1075175
BC00340=131751,862217,1075175
BC00341=131751,862217,1075175
BC00342=131751,862217,1075175
BC00343=131751,862217,1075175
BC00344=107480,867622,1075175
BC00345=36182,883500,1075175
BC00346=36182,883500,1075175
BC00347=36182,883500,1075175
BC00348=36182,883500,1075175
BC00349=36182,883500,1075175
BC00350=36182,883500,1075175
BC00351=36182,883500,1075175
BC00352=36182,883500,1075175
BC00353=36182,883500,1075175
BC00354=36182,883500,1075175
BC00355=65366,862824,1075175
BC00356=79958,852485,1075175
BC00357=79958,852485,1075175
BC00358=79958,852485,1075175
BC00359=79958,852485,1075175
BC00360=79958,852485,1075175
BC00361=79958,852485,1075175
BC00362=79958,852485,1075175
BC00363=79958,852485,1075175
BC00364=79958,852485,1075175
BC00365=79958,852485,1075175
BC00366=79958,852485,1075175
BC00367=79958,852485,1075175
BC00368=79958,852485,1075175
BC00369=253095,795778,1075175
BC00370=253095,795778,1075175
BC00371=253095,795778,1075175
BC00372=253095,795778,1075175
BC00373=253095,795778,1075175
BC00374=253095,795778,1075175
BC00375=253095,795778,1075175
BC00376=253095,795778,1075175
BC00377=253095,795778,1075175
BC00378=253095,795778,1075175
BC00379=253095,795778,1075175
BC00380=277970,773099,1075175
BC00381=277970,773099,1075175
BC00382=277970,773099,1075175
BC00383=277970,773099,1075175
BC00384=277970,773099,1075175
BC00385=277970,773099,1075175
BC00386=277970,773099,1075175
BC00387=277970,773099,1075175
BC00388=277970,773099,1075175
BC00389=277970,773099,1075175
BC00390=277970,773099,1075175
BC00391=277970,773099,1075175
BC00392=391401,773564,1075175
BC00393=391401,773564,1075175
BC00394=391401,773564,1075175
BC00395=391401,773564,1075175
BC00396=391401,773564,1075175
BC00397=391401,773564,1075175
BC00398=391401,773564,1075175
BC00399=391401,773564,1075175
BC00400=391401,773564,1075175
BC00401=391401,773564,1075175
BC00402=391279,862949,1075175
BC00403=391279,862949,1075175
BC00404=391279,862949,1075175
BC00405=391279,862949,1075175
BC00406=391279,862949,1075175
BC00407=391279,862949,1075175
BC00408=391279,862949,1075175
BC00409=391279,862949,1075175
BC00410=391279,862949,1075175
BC00411=391279,862949,1075175
BC00412=391279,862949,1075175
BC00413=356671,865533,1075175
BC00414=337474,866966,1075175
BC00415=275808,871571,1075175
BC00416=275808,871571,1075175
BC00417=275808,871571,1075175
BC00418=275808,871571,1075175
BC00419=275808,871571,1075175
BC00420=275808,871571,1075175
BC00421=275808,871571,1075175
BC00422=275808,871571,1075175
BC00423=275808,871571,1075175
BC00424=275808,871571,1075175
BC00425=275808,871571,1075175
BC00426=307223,910718,1075175
BC00427=307223,910718,1075175
BC00428=307223,910718,1075175
BC00429=307223,910718,1075175
BC00430=307223,910718,1075175
BC00431=307223,910718,1075175
BC00432=307223,910718,1075175
BC00433=307223,910718,1075175
BC00434=307223,910718,1075175
BC00435=307223,910718,1075175
BC00436=285896,934777,1075175
BC00437=287314,930132,1075175
BC00438=287881,928273,1075169
BC00439=287881,928274,1075175
BC00440=287881,928274,1075175
BC00441=331662,908320,1075175
BC00442=298889,925540,1075175
BC00443=304335,922407,1075175
BC00444=306243,923246,1075175
BC00445=311013,925342,1075175
BC00446=310992,925340,1075175
BC00447=288951,837561,1075175
BC00448=272420,771727,1075175
BC00449=272441,771729,1075175
BC00450=274912,778521,1075175
BC00451=275901,781238,1075175
BC00452=275901,781238,1075175
BC00453=275901,781238,1075175
BC00454=271752,783389,1075175
BC00455=238445,800873,1075175
BC00456=234327,803060,1075175
BC00457=233339,800343,1075175
BC00458=230868,793551,1075175
BC00459=78008,861005,1075175
BC00460=77769,868446,1075175
BC00461=77674,871423,1075175
BC00462=77674,871423,1075175
BC00463=77674,871423,1075175
BC00464=23886,880099,1075175
BC00465=19182,880858,1075175
BC00466=19277,877881,1075175
BC00467=19516,870440,1075175
BC00468=19495,870438,1075175
BC00469=326092,855697,1075175
BC00470=326092,855697,1075175
BC00471=398174,852232,1075175
BC00472=398174,857485,1075175
BC00473=398174,859586,1075175
BC00474=398174,859586,1075175
BC00475=398174,859586,1075175
BC00476=371813,869160,1075175
BC00477=367110,869924,1075175
BC00478=367173,867823,1075175
BC00479=367173,867823,1075175
BC00480=367173,867823,1075175
BC00481=360387,856598,1075175
BC00482=311250,775314,1075175
BC00483=310674,772108,1075175
BC00484=310157,770863,1075175
BC00485=310443,770826,1075175
BC00486=310443,770826,1075175
BC00487=310157,770863,1075175
BC00488=281252,771527,1075175
BC00489=281201,772763,1075175
BC00490=283941,775788,1075175
BC00491=283920,775786,1075175
BC00492=277373,824158,1075175
BC00493=275378,838906,1075175
BC00494=277972,845384,1075175
BC00495=279902,846207,1075175
BC00496=279010,847975,1075175
BC00497=279010,847975,1075175
BC00498=308125,844091,1075175
BC00499=270491,850162,1075175
BC00500=273128,849737,1075175
BC00501=273830,846973,1075175
BC00502=275584,840064,1075175
BC00503=275563,840061,1075175
BC00504=324608,813796,1075175
BC00505=398174,774398,1075175
BC00506=398174,774401,1075175
BC00507=398174,771767,1075175
BC00508=398174,771517,1075173
BC00509=398174,770713,1075175
BC00510=398174,770713,1075175
BC00511=345888,773938,1075175
BC00512=391446,773901,1075175
BC00513=395311,773894,1075175
BC00514=395311,773894,1075175
BC00515=395554,778391,1075175
BC00516=395533,778388,1075175
BC00517=244947,801075,1075175
BC00518=66752,827920,1075175
BC00519=66773,827923,1075175
BC00520=63808,834893,1075175
BC00521=62622,837682,1075175
BC00522=62622,837682,1075175
BC00523=62622,837682,1075175
BC00524=65024,838688,1075175
BC00525=67719,839810,1075175
BC00526=67719,839810,1075175
BC00527=71870,830051,1075175
BC00528=97426,846419,1075175
BC00529=97270,849222,1075175
BC00530=97270,849222,1075175
BC00531=97270,849222,1075175
BC00532=92568,849992,1075175
BC00533=61997,854937,1075175
BC00534=64634,854514,1075175
BC00535=65336,851751,1075175
BC00536=84699,851770,1075175
BC00537=124914,851811,1075175
BC00538=124935,851814,1075175
BC00539=122737,858395,1075175
BC00540=121858,861028,1075175
BC00541=121858,861028,1075175
BC00542=121858,861028,1075175
BC00543=124620,862466,1075175
BC00544=125499,859833,1075175
BC00545=127697,853251,1075175
BC00546=127676,853249,1075175
BC00547=204722,814942,1075175
BC00548=204743,814944,1075175
BC00549=206674,821646,1075175
BC00550=207446,824327,1075175
BC00551=207446,824327,1075175
BC00552=207446,824327,1075175
BC00553=204611,825752,1075175
BC00554=203320,826401,1075175
BC00555=200485,827827,1075175
BC00556=199712,825146,1075175
BC00557=197782,818445,1075175
BC00558=159365,837791,1075175
BC00559=161435,844430,1075175
BC00560=162263,847086,1075175
BC00561=162263,847086,1075175
BC00562=162263,847086,1075175
BC00563=158269,849138,1075175
BC00564=157441,846482,1075175
BC00565=155371,839843,1075175
BC00566=121548,857305,1075175
BC00567=123718,863898,1075175
BC00568=124587,866535,1075175
BC00569=124587,866535,1075175
BC00570=124587,866535,1075175
BC00571=120591,868620,1075175
BC00572=119723,865983,1075175
BC00573=117552,859390,1075175
BC00574=117531,859387,1075175
BC00575=246992,896371,1075175
BC00576=220074,877634,1075175
BC00577=181712,850933,1075175
BC00578=181712,850933,1075175
BC00579=238846,900446,1075175
BC00580=238846,900446,1075175
BC00581=233667,887804,1075175
BC00582=233736,914980,1075175
BC00583=230071,889541,1075175
BC00584=233789,896183,1075175
BC00585=229861,888764,1075175
BC00586=221340,873628,1075175
BC00587=204000,858703,1075175
BC00588=181712,850933,1075175
BC00589=163054,850862,1075175
BC00590=145387,858647,1075175
BC00591=143913,859593,1075175
BC00592=142936,860330,1075175
BC00593=147400,860834,1075175
BC00594=147400,860834,1075175
BC00595=147400,860834,1075175
BC00596=147209,858034,1075175
BC00597=146826,852434,1075175
BC00598=162823,738758,1075175
BC00599=162823,738758,1075175
BC00600=162823,738758,1075175
BC00601=162469,668315,1065860
BC00602=132836,722637,395133
BC00603=132836,785697,289538
BC00604=120112,840943,355403
BC00605=120112,840943,355403
BC00606=120112,840943,355403
BC00607=120112,840943,355403
BC00608=120112,840943,355403
BC00609=120112,840943,355403
BC00610=120112,840943,355403
BC00611=120112,840943,355403
BC00612=120112,840943,355403
BC00613=120112,840943,355403
BC00614=112990,845108,322924
BC00615=112990,845108,322924
BC00616=112990,845108,322924
BC00617=112990,845108,322924
BC00618=112990,845108,322924
BC00619=112990,845108,322924
BC00620=112990,845108,322924
BC00621=112990,845108,322924
BC00622=104813,823501,393324
BC00623=104813,823501,393324
BC00624=104813,760081,393324
BC00625=248254,760081,393324
BC00626=248246,711751,217199
BC00627=248240,678922,53
BC00628=292488,813118,262788
BC00629=292488,813118,262788
BC00630=292487,813119,262787
BC00631=292488,813118,262788
BC00632=292488,813118,262788
BC00633=292487,813119,262787
BC00634=292487,813119,262787
BC00635=292487,813119,262787
BC00636=292487,813119,262787
BC00637=292487,813119,262787
BC00638=292488,813118,262788
BC00639=292488,813118,262788
BC00640=292488,813118,262788
BC00641=274061,782472,233150
BC00642=216295,686398,140238
BC00643=267150,771347,84751
BC00644=267150,771347,84751
BC00645=267150,771347,84751
BC00646=267149,771347,84748
BC00647=267150,771347,84751
BC00648=267150,771347,84751
BC00649=267149,771347,84748
BC00650=267149,771347,84748
BC00651=267149,771347,84748
BC00652=267149,771347,84748
BC00653=267149,771347,84748
BC00654=267149,771347,84748
BC00655=267150,771347,84751
BC00656=267150,771347,84751
BC00657=279279,807263,15856
BC00658=279279,807263,15856
BC00659=278551,787027,4009
BC00660=278532,787019,4021
BC00661=278532,787020,4020
BC00662=278532,787020,4020
BC00663=278532,787020,4020
BC00664=278532,787020,4020
BC00665=278532,787020,4020
BC00666=278532,787020,4020
BC00667=278532,787020,4020
BC00668=278532,787020,4020
BC00669=278532,787020,4020
BC00670=278532,787020,4020
BC00671=278532,787020,4020
BC00672=248348,722947,225922
BC00673=227130,668325,385240
BC00674=89228,669140,483629
BC00675=85891,769521,393324
BC00676=85891,823501,393324
BC00677=78694,819217,285317
BC00678=80911,824247,266429
BC00679=81798,826258,258874
BC00680=81798,826258,258874
BC00681=81798,826258,258874
BC00682=77667,828574,258907
BC00683=73118,831123,258944
BC00684=68987,833438,258977
BC00685=68100,831426,266531
BC00686=65882,826396,285419
BC00687=89795,837211,285494
BC00688=92010,842241,266606
BC00689=92896,844254,259052
BC00690=92896,844254,259052
BC00691=92896,844254,259052
BC00692=92896,844254,259052
BC00693=92896,844254,259052
BC00694=92896,844254,259052
BC00695=85891,823501,393324
BC00696=85891,764660,393324
BC00697=85891,709426,393324
BC00698=162291,708666,208254
BC00699=248240,707811,53
BC00700=248240,740511,53
BC00701=263228,763657,33242
BC00702=270136,774326,48540
BC00703=270136,774326,48540
BC00704=289480,804199,91375
BC00705=289480,804199,91375
BC00706=270136,774326,48540
BC00707=270136,774326,48540
BC00708=270419,774762,49166
BC00709=268962,774570,99865
BC00710=269143,774832,97699
BC00711=269143,774832,97699
BC00712=271008,780091,86007
BC00713=271008,780091,86007
BC00714=269143,774832,97699
BC00715=269143,774832,97699
BC00716=268098,775090,99700
BC00717=268098,775090,99700
BC00718=268098,775090,99700
BC00719=268098,775090,99700
BC00720=268098,775090,99700
BC00721=268098,775090,99700
BC00722=268098,775090,99700
BC00723=268098,775090,99700
BC00724=268098,775090,99699
BC00725=268098,775090,99699
BC00726=268098,775090,99699
BC00727=268098,775090,99700
BC00728=268098,775090,99700
BC00729=268098,775090,99700
BC00730=268098,775090,99700
BC00731=268098,775090,99700
BC00732=268098,775090,99700
BC00733=268098,775090,99700
BC00734=268098,775090,99700
BC00735=268098,775090,99700
BC00736=268098,775090,99700
BC00737=268098,775090,99700
BC00738=268098,775090,99700
BC00739=268098,775090,99700
BC00740=268098,775090,99700
BC00741=268098,775090,99700
BC00742=248240,678922,53
BC00743=248240,678922,53
BC00744=325149,799380,131072
BC00745=325149,799380,131072
BC00746=325149,799379,131071
BC00747=325149,799380,131072
BC00748=325149,799380,131072
BC00749=325149,799379,131071
BC00750=325149,799379,131071
BC00751=325149,799379,131071
BC00752=325149,799379,131071
BC00753=325149,799379,131071
BC00754=325149,799379,131071
BC00755=325149,799380,131072
BC00756=309454,697955,17856
BC00757=284186,811897,242158
BC00758=284186,811897,242158
BC00759=284186,811897,242158
BC00760=284186,811897,242158
BC00761=284186,811897,242158
BC00762=284186,811897,242158
BC00763=284186,811897,242158
BC00764=284186,811897,242158
BC00765=294965,806037,143387
BC00766=294965,806037,143387
BC00767=294965,806037,143387
BC00768=294965,806037,143387
BC00769=294965,806037,143387
BC00770=294965,806037,143387
BC00771=294965,806037,143387
BC00772=294965,806037,143387
BC00773=294965,806037,143387
BC00774=346884,805648,147012
BC00775=344714,817518,131657
BC00776=344714,817518,131657
BC00777=344714,817518,131657
BC00778=344714,817518,131657
BC00779=344714,817518,131657
BC00780=344714,817518,131657
BC00781=344714,817518,131657
BC00782=344714,817518,131657
BC00783=344714,817518,131657
BC00784=344714,817518,131657
BC00785=344714,817518,131657
BC00786=289930,764491,131654
BC00787=250055,764491,63495
BC00788=250055,764491,63495
BC00789=250055,764491,63495
BC00790=250055,764491,63495
BC00791=250055,764491,63495
BC00792=250055,764491,63495
BC00793=250055,764491,63492
BC00794=250055,764491,63492
BC00795=250055,764491,63492
BC00796=250055,764491,63492
BC00797=289930,764491,131654
BC00798=344714,668458,131654
BC00799=142431,668458,131654
EC00000=798156,1112951
EC00001=798156,1112951
EC00002=798156,1112951
EC00003=798156,1112951
EC00004=798155,1112951
EC00005=798155,1112951
EC00006=798155,1112951
EC00007=798154,1112950
EC00008=798154,1112950
EC00009=798154,1112950
EC00010=798154,1112950
EC00011=798154,1112950
EC00012=798154,1112950
EC00013=798154,1112950
EC00014=798154,1112950
EC00015=798154,1112950
EC00016=798154,1112950
EC00017=798154,1112950
EC00018=798154,1112950
EC00019=798154,1112950
EC00020=798154,1112950
EC00021=798154,1112950
EC00022=798154,1112950
EC00023=798154,1112950
EC00024=798154,1112950
EC00025=798154,1112950
EC00026=798154,1112950
EC00027=798154,1112950
EC00028=798154,1112950
EC00029=798154,1112950
EC00030=798154,1112950
EC00031=798154,1112950
EC00032=798154,1112950
EC00033=798154,1112950
EC00034=798152,1112949
EC00035=798152,1112949
EC00036=798152,1112949
EC00037=798152,1112949
EC00038=798152,1112949
EC00039=798152,1112949
EC00040=798152,1112949
EC00041=798156,1112951
EC00042=798156,1112951
EC00043=798155,1112951
EC00044=798155,1112951
EC00045=798155,1112951
EC00046=798155,1112951
EC00047=798155,1112951
EC00048=798155,1112951
EC00049=798155,1112951
EC00050=798155,1112951
EC00051=798155,1112951
EC00052=798155,1112951
EC00053=798155,1112951
EC00054=798155,1112951
EC00055=798155,1112951
EC00056=798155,1112951
EC00057=798155,1112951
EC00058=798155,1112951
EC00059=798155,1112951
EC00060=798155,1112951
EC00061=798155,1112951
EC00062=798155,1112951
EC00063=798155,1112951
EC00064=798153,1112950
EC00065=798151,1112948
EC00066=798151,1112948
EC00067=798149,1112947
EC00068=798149,1112947
EC00069=798149,1112947
EC00070=798149,1112947
EC00071=798149,1112947
EC00072=798148,1112946
EC00073=798148,1112946
EC00074=798130,1112937
EC00075=798130,1112937
EC00076=798130,1112937
EC00077=798130,1112937
EC00078=798130,1112937
EC00079=798130,1112937
EC00080=798130,1112937
EC00081=798130,1112937
EC00082=798130,1112937
EC00083=798130,1112937
EC00084=798144,1112944
EC00085=798156,1112951
EC00086=798156,1112951
EC00087=798156,1112951
EC00088=798156,1112951
EC00089=798156,1112951
EC00090=798156,1112951
EC00091=798156,1112951
EC00092=798156,1112951
EC00093=798156,1112951
EC00094=798156,1112951
EC00095=798156,1112951
EC00096=798156,1112951
EC00097=798156,1112951
EC00098=798156,1112951
EC00099=798156,1112951
EC00100=798156,1112951
EC00101=798156,1112951
EC00102=798156,1112951
EC00103=798156,1112951
EC00104=798156,1112951
EC00105=798156,1112951
EC00106=798156,1112951
EC00107=798156,1112951
EC00108=798156,1112951
EC00109=798156,1112951
EC00110=798156,1112951
EC00111=798156,1112951
EC00112=798156,1112951
EC00113=798156,1112951
EC00114=798156,1112951
EC00115=798156,1112951
EC00116=798156,1112951
EC00117=798156,1112951
EC00118=798156,1112951
EC00119=798156,1112951
EC00120=798156,1112951
EC00121=798156,1112951
EC00122=798155,1112950
EC00123=798155,1112950
EC00124=798155,1112950
EC00125=798155,1112950
EC00126=798155,1112950
EC00127=798155,1112950
EC00128=798155,1112950
EC00129=798155,1112950
EC00130=798155,1112950
EC00131=798155,1112950
EC00132=798155,1112950
EC00133=798155,1112950
EC00134=798155,1112950
EC00135=798155,1112950
EC00136=798155,1112950
EC00137=798155,1112950
EC00138=798155,1112950
EC00139=798155,1112950
EC00140=798154,1112950
EC00141=798155,1112950
EC00142=798155,1112950
EC00143=798155,1112950
EC00144=798155,1112950
EC00145=798155,1112950
EC00146=798155,1112950
EC00147=798155,1112950
EC00148=798155,1112950
EC00149=798155,1112950
EC00150=798155,1112950
EC00151=798155,1112950
EC00152=798155,1112950
EC00153=798155,1112950
EC00154=798155,1112950
EC00155=798154,1112949
EC00156=798154,1112949
EC00157=798154,1112949
EC00158=798154,1112949
EC00159=798154,1112949
EC00160=798154,1112949
EC00161=798154,1112949
EC00162=798154,1112949
EC00163=798154,1112949
EC00164=798153,1112947
EC00165=798153,1112947
EC00166=798153,1112947
EC00167=798153,1112947
EC00168=798153,1112947
EC00169=798153,1112947
EC00170=798153,1112947
EC00171=798153,1112947
EC00172=798153,1112947
EC00173=798153,1112947
EC00174=798153,1112947
EC00175=798153,1112947
EC00176=798153,1112947
EC00177=798153,1112947
EC00178=798153,1112947
EC00179=798153,1112947
EC00180=798153,1112947
EC00181=798153,1112947
EC00182=798153,1112947
EC00183=798153,1112947
EC00184=798153,1112947
EC00185=798153,1112947
EC00186=798153,1112947
EC00187=798153,1112947
EC00188=798153,1112947
EC00189=798153,1112947
EC00190=798153,1112947
EC00191=798153,1112947
EC00192=798153,1112947
EC00193=798153,1112947
EC00194=798153,1112947
EC00195=798152,1112946
EC00196=798152,1112946
EC00197=798152,1112946
EC00198=798152,1112946
EC00199=798152,1112946
EC00200=798152,1112946
EC00201=798152,1112946
EC00202=798152,1112946
EC00203=798152,1112946
EC00204=798152,1112946
EC00205=798152,1112946
EC00206=798152,1112946
EC00207=798152,1112946
EC00208=798152,1112946
EC00209=798152,1112946
EC00210=798152,1112946
EC00211=798152,1112946
EC00212=798152,1112946
EC00213=798152,1112946
EC00214=798152,1112946
EC00215=798152,1112946
EC00216=798152,1112946
EC00217=798152,1112946
EC00218=798152,1112946
EC00219=798152,1112946
EC00220=798152,1112946
EC00221=798152,1112946
EC00222=798152,1112946
EC00223=798152,1112946
EC00224=798152,1112946
EC00225=798152,1112946
EC00226=798152,1112946
EC00227=798152,1112946
EC00228=798151,1112945
EC00229=798149,1112944
EC00230=798148,1112944
EC00231=798149,1112944
EC00232=798149,1112944
EC00233=798149,1112944
EC00234=798149,1112944
EC00235=798153,1112947
EC00236=798153,1112947
EC00237=798152,1112946
EC00238=798152,1112946
EC00239=798152,1112946
EC00240=798152,1112946
EC00241=798152,1112946
EC00242=798152,1112946
EC00243=798152,1112946
EC00244=798152,1112946
EC00245=798152,1112946
EC00246=798152,1112946
EC00247=798152,1112946
EC00248=798152,1112946
EC00249=798151,1112945
EC00250=798151,1112945
EC00251=798151,1112945
EC00252=798151,1112945
EC00253=798151,1112945
EC00254=798151,1112945
EC00255=798152,1112946
EC00256=798152,1112946
EC00257=798152,1112946
EC00258=798152,1112946
EC00259=798152,1112946
EC00260=798152,1112946
EC00261=798152,1112946
EC00262=798152,1112946
EC00263=798152,1112946
EC00264=798152,1112946
EC00265=798152,1112946
EC00266=798152,1112946
EC00267=798152,1112946
EC00268=798154,1112949
EC00269=798154,1112949
EC00270=798153,1112947
EC00271=798153,1112947
EC00272=798153,1112947
EC00273=798153,1112947
EC00274=798153,1112947
EC00275=798153,1112947
EC00276=798153,1112947
EC00277=798153,1112947
EC00278=798153,1112947
EC00279=798153,1112947
EC00280=798153,1112947
EC00281=798153,1112947
EC00282=798153,1112947
EC00283=798153,1112947
EC00284=798153,1112947
EC00285=798153,1112947
EC00286=798153,1112947
EC00287=798153,1112947
EC00288=798153,1112947
EC00289=798153,1112947
EC00290=798152,1112946
EC00291=798152,1112946
EC00292=975524,1112951
EC00293=975524,1112951
EC00294=975524,1112951
EC00295=975524,1112951
EC00296=975524,1112951
EC00297=975524,1112951
EC00298=975524,1112951
EC00299=975524,1112951
EC00300=975524,1112951
EC00301=975524,1112951
EC00302=975524,1112951
EC00303=975524,1112951
EC00304=975524,1112951
EC00305=975524,1112951
EC00306=975524,1112951
EC00307=975524,1112951
EC00308=975524,1112951
EC00309=975524,1112951
EC00310=975524,1112951
EC00311=975524,1112951
EC00312=975524,1112951
EC00313=975524,1112951
EC00314=975524,1112951
EC00315=975524,1112951
EC00316=975524,1112951
EC00317=975524,1112951
EC00318=975524,1112951
EC00319=975524,1112951
EC00320=975524,1112951
EC00321=975524,1112951
EC00322=975524,1112951
EC00323=975524,1112951
EC00324=975524,1112951
EC00325=975524,1112951
EC00326=975524,1112951
EC00327=975524,1112951
EC00328=975524,1112951
EC00329=975524,1112951
EC00330=975524,1112951
EC00331=975524,1112951
EC00332=975524,1112951
EC00333=975524,1112951
EC00334=975524,1112951
EC00335=975524,1112951
EC00336=975524,1112951
EC00337=975524,1112951
EC00338=975524,1112951
EC00339=975524,1112951
EC00340=975524,1112951
EC00341=975524,1112951
EC00342=975524,1112951
EC00343=975524,1112951
EC00344=975524,1112951
EC00345=975524,1112951
EC00346=975524,1112951
EC00347=975524,1112951
EC00348=975524,1112951
EC00349=975524,1112951
EC00350=975524,1112951
EC00351=975524,1112951
EC00352=975524,1112951
EC00353=975524,1112951
EC00354=975524,1112951
EC00355=975524,1112951
EC00356=975524,1112951
EC00357=975524,1112951
EC00358=975524,1112951
EC00359=975524,1112951
EC00360=975524,1112951
EC00361=975524,1112951
EC00362=975524,1112951
EC00363=975524,1112951
EC00364=975524,1112951
EC00365=975524,1112951
EC00366=975524,1112951
EC00367=975524,1112951
EC00368=975524,1112951
EC00369=975524,1112951
EC00370=975524,1112951
EC00371=975524,1112951
EC00372=975524,1112951
EC00373=975524,1112951
EC00374=975524,1112951
EC00375=975524,1112951
EC00376=975524,1112951
EC00377=975524,1112951
EC00378=975524,1112951
EC00379=975524,1112951
EC00380=975524,1112951
EC00381=975524,1112951
EC00382=975524,1112951
EC00383=975524,1112951
EC00384=975524,1112951
EC00385=975524,1112951
EC00386=975524,1112951
EC00387=975524,1112951
EC00388=975524,1112951
EC00389=975524,1112951
EC00390=975524,1112951
EC00391=975524,1112951
EC00392=975524,1112951
EC00393=975524,1112951
EC00394=975524,1112951
EC00395=975524,1112951
EC00396=975524,1112951
EC00397=975524,1112951
EC00398=975524,1112951
EC00399=975524,1112951
EC00400=975524,1112951
EC00401=975524,1112951
EC00402=975524,1112951
EC00403=975524,1112951
EC00404=975524,1112951
EC00405=975524,1112951
EC00406=975524,1112951
EC00407=975524,1112951
EC00408=975524,1112951
EC00409=975524,1112951
EC00410=975524,1112951
EC00411=975524,1112951
EC00412=975524,1112951
EC00413=975524,1112951
EC00414=975524,1112951
EC00415=975524,1112951
EC00416=975524,1112951
EC00417=975524,1112951
EC00418=975524,1112951
EC00419=975524,1112951
EC00420=975524,1112951
EC00421=975524,1112951
EC00422=975524,1112951
EC00423=975524,1112951
EC00424=975524,1112951
EC00425=975524,1112951
EC00426=975524,1112951
EC00427=975524,1112951
EC00428=975524,1112951
EC00429=975524,1112951
EC00430=975524,1112951
EC00431=975524,1112951
EC00432=975524,1112951
EC00433=975524,1112951
EC00434=975524,1112951
EC00435=975524,1112951
EC00436=975524,1112951
EC00437=975524,1112951
EC00438=975518,1112948
EC00439=975524,1112951
EC00440=975524,1112951
EC00441=975524,1112951
EC00442=975524,1112951
EC00443=975524,1112951
EC00444=975524,1112951
EC00445=975524,1112951
EC00446=975524,1112951
EC00447=975524,1112951
EC00448=975524,1112951
EC00449=975524,1112951
EC00450=975524,1112951
EC00451=975524,1112951
EC00452=975524,1112951
EC00453=975524,1112951
EC00454=975524,1112951
EC00455=975524,1112951
EC00456=975524,1112951
EC00457=975524,1112951
EC00458=975524,1112951
EC00459=975524,1112951
EC00460=975524,1112951
EC00461=975524,1112951
EC00462=975524,1112951
EC00463=975524,1112951
EC00464=975524,1112951
EC00465=975524,1112951
EC00466=975524,1112951
EC00467=975524,1112951
EC00468=975524,1112951
EC00469=975524,1112951
EC00470=975524,1112951
EC00471=975524,1112951
EC00472=975524,1112951
EC00473=975524,1112951
EC00474=975524,1112951
EC00475=975524,1112951
EC00476=975524,1112951
EC00477=975524,1112951
EC00478=975524,1112951
EC00479=975524,1112951
EC00480=975524,1112951
EC00481=975524,1112951
EC00482=975524,1112951
EC00483=975524,1112951
EC00484=975524,1112951
EC00485=975524,1112951
EC00486=975524,1112951
EC00487=975524,1112951
EC00488=975524,1112951
EC00489=975524,1112951
EC00490=975524,1112951
EC00491=975524,1112951
EC00492=975524,1112951
EC00493=975524,1112951
EC00494=975524,1112951
EC00495=975524,1112951
EC00496=975524,1112951
EC00497=975524,1112951
EC00498=975524,1112951
EC00499=975524,1112951
EC00500=975524,1112951
EC00501=975524,1112951
EC00502=975524,1112951
EC00503=975524,1112951
EC00504=975524,1112951
EC00505=975524,1112951
EC00506=975524,1112951
EC00507=975524,1112951
EC00508=975522,1112950
EC00509=975524,1112951
EC00510=975524,1112951
EC00511=975524,1112951
EC00512=975524,1112951
EC00513=975524,1112951
EC00514=975524,1112951
EC00515=975524,1112951
EC00516=975524,1112951
EC00517=975524,1112951
EC00518=975524,1112951
EC00519=975524,1112951
EC00520=975524,1112951
EC00521=975524,1112951
EC00522=975524,1112951
EC00523=975524,1112951
EC00524=975524,1112951
EC00525=975524,1112951
EC00526=975524,1112951
EC00527=975524,1112951
EC00528=975524,1112951
EC00529=975524,1112951
EC00530=975524,1112951
EC00531=975524,1112951
EC00532=975524,1112951
EC00533=975524,1112951
EC00534=975524,1112951
EC00535=975524,1112951
EC00536=975524,1112951
EC00537=975524,1112951
EC00538=975524,1112951
EC00539=975524,1112951
EC00540=975524,1112951
EC00541=975524,1112951
EC00542=975524,1112951
EC00543=975524,1112951
EC00544=975524,1112951
EC00545=975524,1112951
EC00546=975524,1112951
EC00547=975524,1112951
EC00548=975524,1112951
EC00549=975524,1112951
EC00550=975524,1112951
EC00551=975524,1112951
EC00552=975524,1112951
EC00553=975524,1112951
EC00554=975524,1112951
EC00555=975524,1112951
EC00556=975524,1112951
EC00557=975524,1112951
EC00558=975524,1112951
EC00559=975524,1112951
EC00560=975524,1112951
EC00561=975524,1112951
EC00562=975524,1112951
EC00563=975524,1112951
EC00564=975524,1112951
EC00565=975524,1112951
EC00566=975524,1112951
EC00567=975524,1112951
EC00568=975524,1112951
EC00569=975524,1112951
EC00570=975524,1112951
EC00571=975524,1112951
EC00572=975524,1112951
EC00573=975524,1112951
EC00574=975524,1112951
EC00575=975524,1112951
EC00576=975524,1112951
EC00577=975524,1112951
EC00578=975524,1112951
EC00579=975524,1112951
EC00580=975524,1112951
EC00581=975524,1112951
EC00582=975524,1112951
EC00583=975524,1112951
EC00584=975524,1112951
EC00585=975524,1112951
EC00586=975524,1112951
EC00587=975524,1112951
EC00588=975524,1112951
EC00589=975524,1112951
EC00590=975524,1112951
EC00591=975524,1112951
EC00592=975524,1112951
EC00593=975524,1112951
EC00594=975524,1112951
EC00595=975524,1112951
EC00596=975524,1112951
EC00597=975524,1112951
EC00598=975524,1112951
EC00599=798156,1112951
EC00600=798156,1112951
EC00601=798154,1112951
EC00602=798156,1112951
EC00603=798156,1112951
EC00604=798156,1112951
EC00605=798156,1112951
EC00606=798156,1112951
EC00607=798156,1112951
EC00608=798156,1112951
EC00609=798156,1112951
EC00610=798156,1112951
EC00611=798156,1112951
EC00612=798156,1112951
EC00613=798156,1112951
EC00614=798156,1112951
EC00615=798156,1112951
EC00616=798156,1112951
EC00617=798156,1112951
EC00618=798156,1112951
EC00619=798156,1112951
EC00620=798156,1112951
EC00621=798156,1112951
EC00622=798156,1112951
EC00623=798156,1112951
EC00624=798156,1112951
EC00625=798156,1112951
EC00626=798156,1112951
EC00627=798156,1112951
EC00628=798156,1112951
EC00629=798156,1112951
EC00630=798155,1112950
EC00631=798156,1112951
EC00632=798156,1112951
EC00633=798155,1112950
EC00634=798155,1112950
EC00635=798155,1112950
EC00636=798155,1112950
EC00637=798155,1112950
EC00638=798156,1112951
EC00639=798156,1112951
EC00640=798156,1112951
EC00641=798156,1112951
EC00642=798156,1112951
EC00643=798156,1112951
EC00644=798156,1112951
EC00645=798156,1112951
EC00646=798155,1112949
EC00647=798156,1112951
EC00648=798156,1112951
EC00649=798155,1112949
EC00650=798155,1112949
EC00651=798155,1112949
EC00652=798155,1112949
EC00653=798155,1112949
EC00654=798155,1112949
EC00655=798156,1112951
EC00656=798156,1112951
EC00657=798156,1112951
EC00658=798156,1112951
EC00659=798151,1112948
EC00660=798150,1112623
EC00661=798149,1112622
EC00662=798149,1112622
EC00663=798149,1112622
EC00664=798149,1112622
EC00665=798149,1112622
EC00666=798149,1112622
EC00667=798149,1112622
EC00668=798149,1112622
EC00669=798149,1112622
EC00670=798149,1112622
EC00671=798149,1112622
EC00672=798156,1112951
EC00673=798156,1112951
EC00674=798156,1112951
EC00675=798156,1112951
EC00676=798156,1112951
EC00677=798156,1112951
EC00678=798156,1112951
EC00679=798156,1112951
EC00680=798156,1112951
EC00681=798156,1112951
EC00682=798156,1112951
EC00683=798156,1112951
EC00684=798156,1112951
EC00685=798156,1112951
EC00686=798156,1112951
EC00687=798156,1112951
EC00688=798156,1112951
EC00689=798156,1112951
EC00690=798156,1112951
EC00691=798156,1112951
EC00692=798156,1112951
EC00693=798156,1112951
EC00694=798156,1112951
EC00695=798156,1112951
EC00696=798156,1112951
EC00697=798156,1112951
EC00698=798156,1112951
EC00699=798156,1112951
EC00700=798156,1112951
EC00701=798156,1112951
EC00702=798155,1112950
EC00703=798155,1112950
EC00704=798156,1112951
EC00705=798156,1112951
EC00706=798155,1112950
EC00707=798155,1112950
EC00708=798155,1112950
EC00709=798155,1112950
EC00710=798155,1112950
EC00711=798155,1112950
EC00712=798156,1112951
EC00713=798156,1112951
EC00714=798155,1112950
EC00715=798155,1112950
EC00716=798155,1112950
EC00717=798155,1112950
EC00718=798155,1112950
EC00719=798155,1112950
EC00720=798155,1112950
EC00721=798155,1112950
EC00722=798155,1112950
EC00723=798155,1112950
EC00724=798154,1112949
EC00725=798154,1112949
EC00726=798154,1112949
EC00727=798155,1112950
EC00728=798155,1112950
EC00729=798155,1112950
EC00730=798155,1112950
EC00731=798155,1112950
EC00732=798155,1112950
EC00733=798155,1112950
EC00734=798155,1112950
EC00735=798155,1112950
EC00736=798155,1112950
EC00737=798155,1112950
EC00738=798155,1112950
EC00739=798155,1112950
EC00740=798155,1112950
EC00741=798155,1112950
EC00742=798156,1112951
EC00743=798156,1112951
EC00744=798156,1112951
EC00745=798156,1112951
EC00746=798154,1112949
EC00747=798156,1112951
EC00748=798156,1112951
EC00749=798154,1112949
EC00750=798154,1112949
EC00751=798154,1112949
EC00752=798154,1112949
EC00753=798154,1112949
EC00754=798154,1112949
EC00755=798156,1112951
EC00756=798156,1112951
EC00757=798156,1112951
EC00758=798156,1112951
EC00759=798156,1112951
EC00760=798156,1112951
EC00761=798156,1112951
EC00762=798156,1112951
EC00763=798156,1112951
EC00764=798156,1112951
EC00765=798156,1112951
EC00766=798156,1112951
EC00767=798156,1112951
EC00768=798156,1112951
EC00769=798156,1112951
EC00770=798156,1112951
EC00771=798156,1112951
EC00772=798156,1112951
EC00773=798156,1112951
EC00774=798156,1112951
EC00775=798156,1112951
EC00776=798156,1112951
EC00777=798156,1112951
EC00778=798156,1112951
EC00779=798156,1112951
EC00780=798156,1112951
EC00781=798156,1112951
EC00782=798156,1112951
EC00783=798156,1112951
EC00784=798156,1112951
EC00785=798156,1112951
EC00786=798155,1112950
EC00787=798155,1112950
EC00788=798155,1112950
EC00789=798155,1112950
EC00790=798155,1112950
EC00791=798155,1112950
EC00792=798155,1112950
EC00793=798154,1112950
EC00794=798154,1112950
EC00795=798154,1112950
EC00796=798154,1112950
EC00797=798155,1112950
EC00798=798155,1112950
EC00799=798155,1112950
///POSTYPE BASE
///RECTAN
///RCONF 0,0,0,0,0,0,0,0,0,0,0,0,0,0,0,0,0,0,0,0,0,0,0,0
P00006=0.222,-3.123,-1.508,0.0000,0.0000,0.0000
P00021=-0.225,-6.128,-0.405,0.0000,0.0000,0.0000
P00022=0.222,-3.123,-1.508,0.0000,0.0000,0.0000
P00023=0.143,-0.036,0.682,0.0000,0.0000,0.0000
P00024=0.145,-0.552,1.326,0.0000,0.0000,0.0000
P00025=-2.003,0.006,0.728,0.0000,0.0000,0.0000
P00026=0.562,-0.002,-0.337,0.0000,0.0000,0.0000
P00027=-0.746,0.015,-9.096,0.0000,0.0000,0.0000
P00028=-2.237,-0.018,-7.702,0.0000,0.0000,0.0000
P00029=-2.156,-0.086,-4.681,0.0000,0.0000,0.0000
P00030=5.926,-4.294,-1.390,0.0000,0.0000,0.0000
P00031=1.853,-0.001,-1.549,0.0000,0.0000,0.0000
P00032=1.957,0.503,-7.217,0.0000,0.0000,0.0000
///RCONF 0,0,0,0,1,0,0,0,0,0,0,0,0,0,0,0,0,0,0,0,0,0,0,0
P00033=-0.123,0.612,-5.012,0.0000,0.0000,0.0000
///RCONF 0,0,0,0,0,0,0,0,0,0,0,0,0,0,0,0,0,0,0,0,0,0,0,0
P00034=-0.304,0.773,-2.693,0.0000,0.0000,0.0000
P00035=2.817,0.591,-1.622,0.0000,0.0000,0.0000
P00036=-1.108,-0.829,1.850,0.0000,0.0000,0.0000
P00037=0.023,0.937,-2.677,0.0000,0.0000,0.0000
P00038=0.158,-1.133,-1.952,0.0000,0.0000,0.0000
P00039=0.012,-3.081,-0.106,0.0000,0.0000,0.0000
P00040=-0.030,9.648,2.467,0.0000,0.0000,0.0000
P00041=0.192,3.924,0.305,0.0000,0.0000,0.0000
P00042=-0.217,1.941,0.413,0.0000,0.0000,0.0000
P00043=-0.044,-1.937,1.197,0.0000,0.0000,0.0000
P00044=0.687,-2.322,1.156,0.0000,0.0000,0.0000
P00050=4.296,-4.501,-0.826,0.0000,0.0000,0.0000
P00051=0.367,3.892,0.009,0.0000,0.0000,0.0000
//INST
///DATE 2025/05/13 14:51
///ATTR SC,RW
///GROUP1 RB1,BS1
///GROUP2 ST1
NOP
'OK_r2_O38-47,64(1)(90,180)
'Down
MOVJ C00000 BC00000 VJ=100.00  +MOVJ EC00000 VJ=100.00
MOVJ C00001 BC00001 VJ=100.00  +MOVJ EC00001 VJ=100.00
MOVJ C00002 BC00002 VJ=100.00  +MOVJ EC00002 VJ=100.00
MOVJ C00003 BC00003 VJ=100.00  +MOVJ EC00003 VJ=100.00
MOVL C00004 BC00004 V=666.7  +MOVJ EC00004 VJ=100.00
SMOVL C00005 BC00005 V=166.7  +MOVJ EC00005
SREFP 3 C00006 BC00006  +REFP EC00006
CALL JOB:SEARCH-R1-S13D
SET P024 P006
SFTON3D P024
SMOVL C00007 BC00007 V=166.7  +MOVJ EC00007
SREFP 3 C00008 BC00008  +REFP EC00008
CALL JOB:SEARCH-R1-S13D
SET P024 P006
SFTON3D P024
SMOVL C00009 BC00009 V=166.7  +MOVJ EC00009
SMOVL C00010 BC00010 V=166.7  +MOVJ EC00010
SREFP 3 C00011 BC00011  +REFP EC00011
CALL JOB:SEARCH-R1-S13D
SET P024 P006
SFTON3D P024
SMOVL C00012 BC00012 V=166.7  +MOVJ EC00012
MOVL C00013 BC00013 V=666.7  +MOVJ EC00013 VJ=100.00
SMOVL C00014 BC00014 V=166.7  +MOVJ EC00014
SREFP 3 C00015 BC00015  +REFP EC00015
CALL JOB:SEARCH-R1-S13D
SET P025 P006
SFTON3D P025
SMOVL C00016 BC00016 V=166.7  +MOVJ EC00016
SREFP 3 C00017 BC00017  +REFP EC00017
CALL JOB:SEARCH-R1-S13D
SET P025 P006
SFTON3D P025
SMOVL C00018 BC00018 V=166.7  +MOVJ EC00018
SMOVL C00019 BC00019 V=166.7  +MOVJ EC00019
SREFP 3 C00020 BC00020  +REFP EC00020
CALL JOB:SEARCH-R1-S13D
SET P025 P006
SFTON3D P025
SMOVL C00021 BC00021 V=166.7  +MOVJ EC00021
SFTOF3D
MOVL C00022 BC00022 V=666.7  +MOVJ EC00022 VJ=100.00
SMOVL C00023 BC00023 V=166.7  +MOVJ EC00023
SREFP 3 C00024 BC00024  +REFP EC00024
CALL JOB:SEARCH-R1-S13D
SET P026 P006
SFTON3D P026
SMOVL C00025 BC00025 V=166.7  +MOVJ EC00025
SREFP 3 C00026 BC00026  +REFP EC00026
CALL JOB:SEARCH-R1-S13D
SET P026 P006
SFTON3D P026
SMOVL C00027 BC00027 V=166.7  +MOVJ EC00027
SMOVL C00028 BC00028 V=166.7  +MOVJ EC00028
SREFP 3 C00029 BC00029  +REFP EC00029
CALL JOB:SEARCH-R1-S13D
SET P026 P006
SFTON3D P026
SMOVL C00030 BC00030 V=166.7  +MOVJ EC00030
MOVL C00031 BC00031 V=666.7  +MOVJ EC00031 VJ=100.00
SMOVL C00032 BC00032 V=166.7  +MOVJ EC00032
SREFP 3 C00033 BC00033  +REFP EC00033
CALL JOB:SEARCH-R1-S13D
SET P027 P006
SFTON3D P027
SMOVL C00034 BC00034 V=166.7  +MOVJ EC00034
SREFP 3 C00035 BC00035  +REFP EC00035
CALL JOB:SEARCH-R1-S13D
SET P027 P006
SFTON3D P027
SMOVL C00036 BC00036 V=166.7  +MOVJ EC00036
SMOVL C00037 BC00037 V=166.7  +MOVJ EC00037
SREFP 3 C00038 BC00038  +REFP EC00038
CALL JOB:SEARCH-R1-S13D
SET P027 P006
SFTON3D P027
SMOVL C00039 BC00039 V=166.7  +MOVJ EC00039
SFTOF3D
'Path S1883
MOVJ C00040 BC00040 VJ=100.00  +MOVJ EC00040 VJ=100.00
MOVL C00041 BC00041 V=500.0  +MOVJ EC00041 VJ=100.00
MOVL C00042 BC00042 V=500.0  +MOVJ EC00042 VJ=100.00
SMOVL C00043 BC00043 V=100.0  +MOVJ EC00043
SREFP 3 C00044 BC00044  +REFP EC00044
CALL JOB:SEARCH-R1-S13D
SET P028 P006
SFTON3D P028
SMOVL C00045 BC00045 V=100.0  +MOVJ EC00045
SMOVL C00046 BC00046 V=100.0  +MOVJ EC00046
SMOVL C00047 BC00047 V=100.0  +MOVJ EC00047
SREFP 3 C00048 BC00048  +REFP EC00048
CALL JOB:SEARCH-R1-S13D
SET P028 P006
SFTON3D P028
SMOVL C00049 BC00049 V=100.0  +MOVJ EC00049
SREFP 3 C00050 BC00050  +REFP EC00050
CALL JOB:SEARCH-R1-S13D
SET P021 P006
SFTON3D P021
SMOVL C00051 BC00051 V=100.0  +MOVJ EC00051
SMOVL C00052 BC00052 V=100.0  +MOVJ EC00052
SMOVL C00053 BC00053 V=100.0  +MOVJ EC00053
SREFP 3 C00054 BC00054  +REFP EC00054
CALL JOB:SEARCH-R1-S13D
SET P021 P006
SFTON3D P021
SMOVL C00055 BC00055 V=100.0  +MOVJ EC00055
MOVL C00056 BC00056 V=500.0  +MOVJ EC00056 VJ=100.00
SMOVL C00057 BC00057 V=166.7  +MOVJ EC00057
SREFP 3 C00058 BC00058  +REFP EC00058
CALL JOB:SEARCH-R1-S13D
SET P029 P006
SFTON3D P029
SMOVL C00059 BC00059 V=166.7  +MOVJ EC00059
SMOVL C00060 BC00060 V=166.7  +MOVJ EC00060
SMOVL C00061 BC00061 V=166.7  +MOVJ EC00061
SREFP 3 C00062 BC00062  +REFP EC00062
CALL JOB:SEARCH-R1-S13D
SET P029 P006
SFTON3D P029
SMOVL C00063 BC00063 V=166.7  +MOVJ EC00063
SFTOF3D
MOVL C00064 BC00064 V=666.7  +MOVJ EC00064 VJ=100.00
MOVL C00065 BC00065 V=666.7  +MOVJ EC00065 VJ=100.00
MOVL C00066 BC00066 V=666.7  +MOVJ EC00066 VJ=100.00
SMOVL C00067 BC00067 V=166.7  +MOVJ EC00067
SREFP 3 C00068 BC00068  +REFP EC00068
CALL JOB:SEARCH-R1-S13D
SET P050 P006
SFTON3D P050
SMOVL C00069 BC00069 V=166.7  +MOVJ EC00069
SREFP 3 C00070 BC00070  +REFP EC00070
CALL JOB:SEARCH-R1-S13D
SET P050 P006
SFTON3D P050
SMOVL C00071 BC00071 V=166.7  +MOVJ EC00071
SMOVL C00072 BC00072 V=166.7  +MOVJ EC00072
SREFP 3 C00073 BC00073  +REFP EC00073
CALL JOB:SEARCH-R1-S13D
SET P050 P006
SFTON3D P050
SMOVL C00074 BC00074 V=166.7  +MOVJ EC00074
MOVL C00075 BC00075 V=666.7  +MOVJ EC00075 VJ=100.00
SMOVL C00076 BC00076 V=166.7  +MOVJ EC00076
SREFP 3 C00077 BC00077  +REFP EC00077
CALL JOB:SEARCH-R1-S13D
SET P051 P006
SFTON3D P051
SMOVL C00078 BC00078 V=166.7  +MOVJ EC00078
SREFP 3 C00079 BC00079  +REFP EC00079
CALL JOB:SEARCH-R1-S13D
SET P051 P006
SFTON3D P051
SMOVL C00080 BC00080 V=166.7  +MOVJ EC00080
SMOVL C00081 BC00081 V=166.7  +MOVJ EC00081
SREFP 3 C00082 BC00082  +REFP EC00082
CALL JOB:SEARCH-R1-S13D
SET P051 P006
SFTON3D P051
SMOVL C00083 BC00083 V=166.7  +MOVJ EC00083
SFTOF3D
MOVL C00084 BC00084 V=400.0  +MOVJ EC00084 VJ=100.00
MOVL C00085 BC00085 V=400.0  +MOVJ EC00085 VJ=100.00
MOVJ C00086 BC00086 VJ=100.00  +MOVJ EC00086 VJ=100.00
MOVJ C00087 BC00087 VJ=100.00  +MOVJ EC00087 VJ=100.00
MOVJ C00088 BC00088 VJ=100.00  +MOVJ EC00088 VJ=100.00
MOVJ C00089 BC00089 VJ=100.00  +MOVJ EC00089 VJ=100.00
'Path S1884
SFTOF3D
MOVJ C00090 BC00090 VJ=40.00  +MOVJ EC00090 VJ=100.00
MOVL C00091 BC00091 V=400.0  +MOVJ EC00091 VJ=100.00
SMOVL C00092 BC00092 V=100.0  +MOVJ EC00092
SREFP 3 C00093 BC00093  +REFP EC00093
CALL JOB:SEARCH-R1-S13D
SET P022 P006
SFTON3D P022
SMOVL C00094 BC00094 V=100.0  +MOVJ EC00094
SMOVL C00095 BC00095 V=133.3  +MOVJ EC00095
SMOVL C00096 BC00096 V=100.0  +MOVJ EC00096
SREFP 3 C00097 BC00097  +REFP EC00097
CALL JOB:SEARCH-R1-S13D
SET P022 P006
SFTON3D P022
SMOVL C00098 BC00098 V=100.0  +MOVJ EC00098
MOVL C00099 BC00099 V=1000.0  +MOVJ EC00099 VJ=100.00
MOVJ C00100 BC00100 VJ=100.00  +MOVJ EC00100 VJ=100.00
MOVJ C00101 BC00101 VJ=100.00  +MOVJ EC00101 VJ=100.00
MOVJ C00102 BC00102 VJ=100.00  +MOVJ EC00102 VJ=100.00
MOVJ C00103 BC00103 VJ=100.00  +MOVJ EC00103 VJ=100.00
MOVJ C00104 BC00104 VJ=100.00  +MOVJ EC00104 VJ=100.00
'Path S1885
SFTOF3D
MOVJ C00105 BC00105 VJ=100.00  +MOVJ EC00105 VJ=100.00
MOVL C00106 BC00106 V=166.7  +MOVJ EC00106 VJ=100.00
SMOVL C00107 BC00107 V=100.0  +MOVJ EC00107
SREFP 3 C00108 BC00108  +REFP EC00108
CALL JOB:SEARCH-R1-S13D
SET P023 P006
SFTON3D P023
SMOVL C00109 BC00109 V=100.0  +MOVJ EC00109
SMOVL C00110 BC00110 V=166.7  +MOVJ EC00110
SMOVL C00111 BC00111 V=100.0  +MOVJ EC00111
SREFP 3 C00112 BC00112  +REFP EC00112
CALL JOB:SEARCH-R1-S13D
SET P023 P006
SFTON3D P023
SMOVL C00113 BC00113 V=100.0  +MOVJ EC00113
SFTOF3D
MOVL C00114 BC00114 V=400.0  +MOVJ EC00114 VJ=100.00
MOVL C00115 BC00115 V=1000.0  +MOVJ EC00115 VJ=100.00
MOVL C00116 BC00116 V=1000.0  +MOVJ EC00116 VJ=100.00
MOVJ C00117 BC00117 VJ=100.00  +MOVJ EC00117 VJ=100.00
MOVJ C00118 BC00118 VJ=100.00  +MOVJ EC00118 VJ=100.00
MOVJ C00119 BC00119 VJ=100.00  +MOVJ EC00119 VJ=100.00
'NOWY PROGRAM KRIS
MOVJ C00120 BC00120 VJ=100.00  +MOVJ EC00120 VJ=100.00
MOVJ C00121 BC00121 VJ=100.00  +MOVJ EC00121 VJ=100.00
MOVJ C00122 BC00122 VJ=100.00  +MOVJ EC00122 VJ=100.00
COMM PAUSE
COMM SMOVL C00123 BC00123 V=100.0  +MOVJ EC00123
COMM SREFP 3 C00124 BC00124  +REFP EC00124
COMM CALL JOB:SEARCH-R1-S13D
COMM SET P030 P006
COMM SFTON3D P030
COMM SMOVL C00125 BC00125 V=100.0  +MOVJ EC00125
COMM SREFP 3 C00126 BC00126  +REFP EC00126
COMM CALL JOB:SEARCH-R1-S13D
COMM SET P030 P006
COMM SFTON3D P030
COMM SMOVL C00127 BC00127 V=100.0  +MOVJ EC00127
COMM SFTOF3D
COMM MOVJ C00128 BC00128 VJ=100.00  +MOVJ EC00128 VJ=100.00
COMM SMOVL C00129 BC00129 V=100.0  +MOVJ EC00129
COMM SREFP 3 C00130 BC00130  +REFP EC00130
COMM CALL JOB:SEARCH-R1-S13D
COMM SET P031 P006
COMM SFTON3D P031
COMM SMOVL C00131 BC00131 V=100.0  +MOVJ EC00131
COMM SREFP 3 C00132 BC00132  +REFP EC00132
COMM CALL JOB:SEARCH-R1-S13D
COMM SET P031 P006
COMM SFTON3D P031
COMM SMOVL C00133 BC00133 V=100.0  +MOVJ EC00133
COMM SFTOF3D
MOVJ C00134 BC00134 VJ=100.00  +MOVJ EC00134 VJ=100.00
MOVJ C00135 BC00135 VJ=100.00  +MOVJ EC00135 VJ=100.00
MOVJ C00136 BC00136 VJ=100.00  +MOVJ EC00136 VJ=100.00
SMOVL C00137 BC00137 V=100.0  +MOVJ EC00137
SREFP 3 C00138 BC00138  +REFP EC00138
CALL JOB:SEARCH-R1-S13D
SET P032 P006
SFTON3D P032
SMOVL C00139 BC00139 V=100.0  +MOVJ EC00139
SREFP 3 C00140 BC00140  +REFP EC00140
CALL JOB:SEARCH-R1-S13D
SET P032 P006
SFTON3D P032
SMOVL C00141 BC00141 V=100.0  +MOVJ EC00141
SFTOF3D
MOVJ C00142 BC00142 VJ=100.00  +MOVJ EC00142 VJ=100.00
SMOVL C00143 BC00143 V=100.0  +MOVJ EC00143
SREFP 3 C00144 BC00144  +REFP EC00144
CALL JOB:SEARCH-R1-S13D
SET P033 P006
SFTON3D P033
SMOVL C00145 BC00145 V=100.0  +MOVJ EC00145
SREFP 3 C00146 BC00146  +REFP EC00146
CALL JOB:SEARCH-R1-S13D
SET P033 P006
SFTON3D P033
SMOVL C00147 BC00147 V=100.0  +MOVJ EC00147
SFTOF3D
MOVJ C00148 BC00148 VJ=100.00  +MOVJ EC00148 VJ=100.00
MOVJ C00149 BC00149 VJ=100.00  +MOVJ EC00149 VJ=100.00
SMOVL C00150 BC00150 V=100.0  +MOVJ EC00150
SREFP 3 C00151 BC00151  +REFP EC00151
CALL JOB:SEARCH-R1-S13D
SET P034 P006
SFTON3D P034
SMOVL C00152 BC00152 V=100.0  +MOVJ EC00152
SREFP 3 C00153 BC00153  +REFP EC00153
CALL JOB:SEARCH-R1-S13D
SET P034 P006
SFTON3D P034
SMOVL C00154 BC00154 V=100.0  +MOVJ EC00154
SFTOF3D
MOVJ C00155 BC00155 VJ=100.00  +MOVJ EC00155 VJ=100.00
MOVJ C00156 BC00156 VJ=100.00  +MOVJ EC00156 VJ=100.00
MOVJ C00157 BC00157 VJ=100.00  +MOVJ EC00157 VJ=100.00
SMOVL C00158 BC00158 V=100.0  +MOVJ EC00158
SREFP 3 C00159 BC00159  +REFP EC00159
CALL JOB:SEARCH-R1-S13D
SET P035 P006
SFTON3D P035
SMOVL C00160 BC00160 V=100.0  +MOVJ EC00160
SREFP 3 C00161 BC00161  +REFP EC00161
CALL JOB:SEARCH-R1-S13D
SET P035 P006
SFTON3D P035
SMOVL C00162 BC00162 V=100.0  +MOVJ EC00162
SFTOF3D
MOVJ C00163 BC00163 VJ=100.00  +MOVJ EC00163 VJ=100.00
SMOVL C00164 BC00164 V=100.0  +MOVJ EC00164
SREFP 3 C00165 BC00165  +REFP EC00165
CALL JOB:SEARCH-R1-S13D
SET P036 P006
SFTON3D P036
SMOVL C00166 BC00166 V=100.0  +MOVJ EC00166
SREFP 3 C00167 BC00167  +REFP EC00167
CALL JOB:SEARCH-R1-S13D
SET P036 P006
SFTON3D P036
SMOVL C00168 BC00168 V=100.0  +MOVJ EC00168
SFTOF3D
MOVJ C00169 BC00169 VJ=100.00  +MOVJ EC00169 VJ=100.00
MOVJ C00170 BC00170 VJ=100.00  +MOVJ EC00170 VJ=100.00
MOVJ C00171 BC00171 VJ=100.00  +MOVJ EC00171 VJ=100.00
SMOVL C00172 BC00172 V=100.0  +MOVJ EC00172
SREFP 3 C00173 BC00173  +REFP EC00173
CALL JOB:SEARCH-R1-S13D
SET P044 P006
SFTON3D P044
SMOVL C00174 BC00174 V=100.0  +MOVJ EC00174
SREFP 3 C00175 BC00175  +REFP EC00175
CALL JOB:SEARCH-R1-S13D
SET P044 P006
SFTON3D P044
SMOVL C00176 BC00176 V=100.0  +MOVJ EC00176
SFTOF3D
MOVJ C00177 BC00177 VJ=100.00  +MOVJ EC00177 VJ=100.00
MOVJ C00178 BC00178 VJ=100.00  +MOVJ EC00178 VJ=100.00
COMM PAUSE
COMM MOVJ C00179 BC00179 VJ=100.00  +MOVJ EC00179 VJ=100.00
COMM MOVJ C00180 BC00180 VJ=100.00  +MOVJ EC00180 VJ=100.00
COMM SMOVL C00181 BC00181 V=100.0  +MOVJ EC00181
COMM SREFP 3 C00182 BC00182  +REFP EC00182
COMM CALL JOB:SEARCH-R1-S13D
COMM SET P037 P006
COMM SFTON3D P037
COMM SMOVL C00183 BC00183 V=100.0  +MOVJ EC00183
COMM SREFP 3 C00184 BC00184  +REFP EC00184
COMM CALL JOB:SEARCH-R1-S13D
COMM SET P037 P006
COMM SFTON3D P037
COMM SMOVL C00185 BC00185 V=100.0  +MOVJ EC00185
COMM SFTOF3D
COMM MOVJ C00186 BC00186 VJ=100.00  +MOVJ EC00186 VJ=100.00
COMM SMOVL C00187 BC00187 V=100.0  +MOVJ EC00187
COMM SREFP 3 C00188 BC00188  +REFP EC00188
COMM CALL JOB:SEARCH-R1-S13D
COMM SET P038 P006
COMM SFTON3D P038
COMM SMOVL C00189 BC00189 V=100.0  +MOVJ EC00189
COMM SREFP 3 C00190 BC00190  +REFP EC00190
COMM CALL JOB:SEARCH-R1-S13D
COMM SET P038 P006
COMM SFTON3D P038
COMM SMOVL C00191 BC00191 V=100.0  +MOVJ EC00191
COMM SFTOF3D
COMM MOVJ C00192 BC00192 VJ=100.00  +MOVJ EC00192 VJ=100.00
MOVJ C00193 BC00193 VJ=100.00  +MOVJ EC00193 VJ=100.00
MOVJ C00194 BC00194 VJ=100.00  +MOVJ EC00194 VJ=100.00
MOVJ C00195 BC00195 VJ=100.00  +MOVJ EC00195 VJ=100.00
SMOVL C00196 BC00196 V=100.0  +MOVJ EC00196
SREFP 3 C00197 BC00197  +REFP EC00197
CALL JOB:SEARCH-R1-S13D
SET P039 P006
SFTON3D P039
SMOVL C00198 BC00198 V=100.0  +MOVJ EC00198
SREFP 3 C00199 BC00199  +REFP EC00199
CALL JOB:SEARCH-R1-S13D
SET P039 P006
SFTON3D P039
SMOVL C00200 BC00200 V=100.0  +MOVJ EC00200
SFTOF3D
MOVJ C00201 BC00201 VJ=100.00  +MOVJ EC00201 VJ=100.00
SMOVL C00202 BC00202 V=100.0  +MOVJ EC00202
SREFP 3 C00203 BC00203  +REFP EC00203
CALL JOB:SEARCH-R1-S13D
SET P040 P006
SFTON3D P040
SMOVL C00204 BC00204 V=100.0  +MOVJ EC00204
SREFP 3 C00205 BC00205  +REFP EC00205
CALL JOB:SEARCH-R1-S13D
SET P040 P006
SFTON3D P040
SMOVL C00206 BC00206 V=100.0  +MOVJ EC00206
MOVJ C00207 BC00207 VJ=100.00  +MOVJ EC00207 VJ=100.00
SFTOF3D
MOVJ C00208 BC00208 VJ=100.00  +MOVJ EC00208 VJ=100.00
MOVJ C00209 BC00209 VJ=100.00  +MOVJ EC00209 VJ=100.00
SMOVL C00210 BC00210 V=100.0  +MOVJ EC00210
SREFP 3 C00211 BC00211  +REFP EC00211
CALL JOB:SEARCH-R1-S13D
SET P041 P006
SFTON3D P041
SMOVL C00212 BC00212 V=100.0  +MOVJ EC00212
SREFP 3 C00213 BC00213  +REFP EC00213
CALL JOB:SEARCH-R1-S13D
SET P041 P006
SFTON3D P041
SMOVL C00214 BC00214 V=100.0  +MOVJ EC00214
SFTOF3D
MOVJ C00215 BC00215 VJ=100.00  +MOVJ EC00215 VJ=100.00
SMOVL C00216 BC00216 V=100.0  +MOVJ EC00216
SREFP 3 C00217 BC00217  +REFP EC00217
CALL JOB:SEARCH-R1-S13D
SET P042 P006
SFTON3D P042
SMOVL C00218 BC00218 V=100.0  +MOVJ EC00218
SREFP 3 C00219 BC00219  +REFP EC00219
CALL JOB:SEARCH-R1-S13D
SET P042 P006
SFTON3D P042
SMOVL C00220 BC00220 V=250.0  +MOVJ EC00220
MOVJ C00221 BC00221 VJ=100.00  +MOVJ EC00221 VJ=100.00
SFTOF3D
MOVJ C00222 BC00222 VJ=100.00  +MOVJ EC00222 VJ=100.00
SMOVL C00223 BC00223 V=100.0  +MOVJ EC00223
SREFP 3 C00224 BC00224  +REFP EC00224
CALL JOB:SEARCH-R1-S13D
SET P043 P006
SFTON3D P043
SMOVL C00225 BC00225 V=100.0  +MOVJ EC00225
SREFP 3 C00226 BC00226  +REFP EC00226
CALL JOB:SEARCH-R1-S13D
SET P043 P006
SFTON3D P043
SMOVL C00227 BC00227 V=166.7  +MOVJ EC00227
'KONIEC POMIARU
SMOVL C00228 BC00228 V=166.7  +MOVJ EC00228
MACRO1 MJ#(0) ARGF9
SFTON3D P043
SMOVL C00229 BC00229 V=250.0  +MOVJ EC00229
ARCON
SWVON WEV#(30)
SMOVL C00230 BC00230 V=10.0  +MOVJ EC00230
SMOVL C00231 BC00231 V=10.0  +MOVJ EC00231
SMOVL C00232 BC00232 V=10.0  +MOVJ EC00232
ARCOF
SWVOF
SFTOF3D
MOVJ C00233 BC00233 VJ=15.00  +MOVJ EC00233 VJ=100.00
MOVJ C00234 BC00234 VJ=100.00  +MOVJ EC00234 VJ=100.00
MOVJ C00235 BC00235 VJ=100.00  +MOVJ EC00235 VJ=100.00
MOVJ C00236 BC00236 VJ=100.00  +MOVJ EC00236 VJ=100.00
SFTON3D P044
SMOVL C00237 BC00237 V=166.7 PL=0  +MOVJ EC00237
ARCON
SWVON WEV#(30)
SMOVL C00238 BC00238 V=8.3  +MOVJ EC00238
SMOVL C00239 BC00239 V=8.3  +MOVJ EC00239
SMOVL C00240 BC00240 V=8.3  +MOVJ EC00240
ARCOF
SWVOF
SFTOF3D
MOVJ C00241 BC00241 VJ=15.00  +MOVJ EC00241 VJ=15.00
COMM PAUSE
COMM MOVJ C00242 BC00242 VJ=100.00  +MOVJ EC00242 VJ=100.00
COMM MACRO1 MJ#(0) ARGF9
COMM SFTON3D P031
COMM SMOVL C00243 BC00243 V=133.3  +MOVJ EC00243
COMM ARCON
COMM SWVON WEV#(10)
COMM SMOVL C00244 BC00244 V=10.0  +MOVJ EC00244
COMM SFTON3D P030
COMM SMOVL C00245 BC00245 V=10.0  +MOVJ EC00245
COMM SMOVL C00246 BC00246 V=10.0  +MOVJ EC00246
COMM ARCOF
COMM SWVOF
COMM SFTOF
COMM MOVJ C00247 BC00247 VJ=100.00  +MOVJ EC00247 VJ=100.00
COMM MOVJ C00248 BC00248 VJ=100.00  +MOVJ EC00248 VJ=100.00
COMM MOVJ C00249 BC00249 VJ=100.00  +MOVJ EC00249 VJ=100.00
COMM SFTON3D P038
COMM SMOVL C00250 BC00250 V=166.7  +MOVJ EC00250
COMM ARCON
COMM SFTON3D P037
COMM MOVL C00251 BC00251 V=9.2  +MOVJ EC00251 VJ=100.00
COMM ARCOF
COMM TIMER T=1.00
COMM SFTOF3D
COMM MOVJ C00252 BC00252 VJ=100.00  +MOVJ EC00252 VJ=100.00
COMM MOVJ C00253 BC00253 VJ=100.00  +MOVJ EC00253 VJ=100.00
COMM MOVJ C00254 BC00254 VJ=100.00  +MOVJ EC00254 VJ=100.00
MOVJ C00255 BC00255 VJ=100.00  +MOVJ EC00255 VJ=100.00
MACRO1 MJ#(0) ARGF14
MOVJ C00256 BC00256 VJ=100.00  +MOVJ EC00256 VJ=100.00
SFTON3D P041
SMOVL C00257 BC00257 V=166.7  +MOVJ EC00257
ARCON
SMOVL C00258 BC00258 V=9.2  +MOVJ EC00258
SFTON3D P042
SMOVL C00259 BC00259 V=9.2  +MOVJ EC00259
ARCOF
SFTOF3D
MOVJ C00260 BC00260 VJ=100.00  +MOVJ EC00260 VJ=100.00
MOVJ C00261 BC00261 VJ=100.00  +MOVJ EC00261 VJ=100.00
SFTON3D P040
SMOVL C00262 BC00262 V=166.7  +MOVJ EC00262
ARCON
SMOVL C00263 BC00263 V=9.2  +MOVJ EC00263
SFTON3D P039
SMOVL C00264 BC00264 V=9.2  +MOVJ EC00264
SMOVL C00265 BC00265 V=9.2  +MOVJ EC00265
ARCOF
MOVJ C00266 BC00266 VJ=100.00  +MOVJ EC00266 VJ=100.00
MOVJ C00267 BC00267 VJ=100.00  +MOVJ EC00267 VJ=100.00
MOVJ C00268 BC00268 VJ=100.00  +MOVJ EC00268 VJ=100.00
MOVJ C00269 BC00269 VJ=100.00  +MOVJ EC00269 VJ=100.00
MACRO1 MJ#(0) ARGF9
SFTON3D P036
SMOVL C00270 BC00270 V=166.7  +MOVJ EC00270
ARCON
SMOVL C00271 BC00271 V=9.2  +MOVJ EC00271
SFTON3D P035
SMOVL C00272 BC00272 V=9.2  +MOVJ EC00272
SMOVL C00273 BC00273 V=9.2  +MOVJ EC00273
ARCOF
SFTOF3D
MOVJ C00274 BC00274 VJ=15.00  +MOVJ EC00274 VJ=100.00
MOVJ C00275 BC00275 VJ=100.00  +MOVJ EC00275 VJ=15.00
MACRO1 MJ#(0) ARGF9
SFTON3D P034
SMOVL C00276 BC00276 V=166.7  +MOVJ EC00276
ARCON
SMOVC C00277 BC00277 V=8.3  +MOVJ EC00277
SMOVC C00278 BC00278 V=8.3  +MOVJ EC00278
SMOVC C00279 BC00279 V=8.3  +MOVJ EC00279
SMOVL C00280 BC00280 V=10.0  +MOVJ EC00280
SMOVC C00281 BC00281 V=8.3  +MOVJ EC00281
SMOVC C00282 BC00282 V=8.3  +MOVJ EC00282
SMOVC C00283 BC00283 V=8.3  +MOVJ EC00283
ARCOF
SFTOF3D
MOVJ C00284 BC00284 VJ=100.00  +MOVJ EC00284 VJ=100.00
MOVJ C00285 BC00285 VJ=100.00  +MOVJ EC00285 VJ=100.00
SFTON3D P032
SMOVL C00286 BC00286 V=250.0  +MOVJ EC00286
ARCON
SMOVL C00287 BC00287 V=8.3  +MOVJ EC00287
SFTON3D P033
SMOVL C00288 BC00288 V=8.3  +MOVJ EC00288
SMOVL C00289 BC00289 V=8.3  +MOVJ EC00289
ARCOF
SFTOF3D
MOVJ C00290 BC00290 VJ=30.00  +MOVJ EC00290 VJ=100.00
MOVJ C00291 BC00291 VJ=30.00  +MOVJ EC00291 VJ=15.00
JUMP *LABEL
'Up
'Path S1856
SFTOF3D
MOVJ C00292 BC00292 VJ=100.00  +MOVJ EC00292 VJ=100.00
COMM MOVL C00293 BC00293 V=400.0  +MOVJ EC00293 VJ=100.00
COMM SMOVL C00294 BC00294 V=60.0  +MOVJ EC00294
COMM SREFP 3 C00295 BC00295  +REFP EC00295
COMM CALL JOB:SEARCH-R1-S13D
COMM SET P042 P006
COMM SFTON3D P042
COMM SMOVL C00296 BC00296 V=60.0  +MOVJ EC00296
COMM SMOVL C00297 BC00297 V=60.0  +MOVJ EC00297
COMM SREFP 3 C00298 BC00298  +REFP EC00298
COMM CALL JOB:SEARCH-R1-S13D
COMM SET P042 P006
COMM SFTON3D P042
COMM SMOVL C00299 BC00299 V=60.0  +MOVJ EC00299
COMM MOVL C00300 BC00300 V=400.0  +MOVJ EC00300 VJ=100.00
COMM MOVL C00301 BC00301 V=1000.0  +MOVJ EC00301 VJ=100.00
COMM 'Path S1857
COMM SFTOF3D
COMM MOVJ C00302 BC00302 VJ=100.00  +MOVJ EC00302 VJ=100.00
COMM MOVL C00303 BC00303 V=400.0  +MOVJ EC00303 VJ=100.00
COMM SMOVL C00304 BC00304 V=60.0  +MOVJ EC00304
COMM SREFP 3 C00305 BC00305  +REFP EC00305
COMM CALL JOB:SEARCH-R1-S13D
COMM SET P041 P006
COMM SFTON3D P041
